LIN {X 0,Y 170.395,Z 400.641,A -85,B 0,C 180,E1 -23240.523,E2 -23240.523} C_VEL
LIN {X 0,Y 173.665,Z 396.703,A -85,B 0,C 180,E1 -23242.047,E2 -23242.047} C_VEL
LIN {X 0,Y 175.029,Z 394.829,A -85,B 0,C 180,E1 -23242.551,E2 -23242.551} C_VEL
LIN {X 0,Y 176.798,Z 393.099,A -85,B 0,C 180,E1 -23243.423,E2 -23243.423} C_VEL
LIN {X 0,Y 178.535,Z 391.866,A -85,B 0,C 180,E1 -23244.414,E2 -23244.414} C_VEL
LIN {X 0,Y 181.801,Z 388.149,A -85,B 0,C 180,E1 -23245.779,E2 -23245.779} C_VEL
LIN {X 0,Y 185.617,Z 382.76,A -85,B 0,C 180,E1 -23247.024,E2 -23247.024} C_VEL
LIN {X 0,Y 188.526,Z 380.586,A -85,B 0,C 180,E1 -23248.379,E2 -23248.379} C_VEL
LIN {X 0,Y 191.312,Z 377.501,A -85,B 0,C 180,E1 -23249.395,E2 -23249.395} C_VEL
LIN {X 0,Y 192.302,Z 378.568,A -85,B 0,C 180,E1 -23250.142,E2 -23250.142} C_VEL
LIN {X 0,Y 194.191,Z 381.489,A -85,B 0,C 180,E1 -23251.653,E2 -23251.653} C_VEL
LIN {X 0,Y 197.755,Z 388.389,A -85,B 0,C 180,E1 -23254.655,E2 -23254.655} C_VEL
LIN {X 0,Y 201.159,Z 397.142,A -85,B 0,C 180,E1 -23257.878,E2 -23257.878} C_VEL
LIN {X 0,Y 202.808,Z 403.388,A -85,B 0,C 180,E1 -23259.875,E2 -23259.875} C_VEL
LIN {X 0,Y 204.423,Z 413.612,A -85,B 0,C 180,E1 -23262.894,E2 -23262.894} C_VEL
LIN {X 0,Y 204.93,Z 420.786,A -85,B 0,C 180,E1 -23264.939,E2 -23264.939} C_VEL
LIN {X 0,Y 203.024,Z 426.169,A -85,B 0,C 180,E1 -23265.89,E2 -23265.89} C_VEL
LIN {X 0,Y 197.868,Z 437.857,A -85,B 0,C 180,E1 -23268.105,E2 -23268.105} C_VEL
LIN {X 0,Y 192.442,Z 449.393,A -85,B 0,C 180,E1 -23270.951,E2 -23270.951} C_VEL
LIN {X 0,Y 187.443,Z 458.742,A -85,B 0,C 180,E1 -23273.805,E2 -23273.805} C_VEL
LIN {X 0,Y 182.067,Z 467.908,A -85,B 0,C 180,E1 -23277.287,E2 -23277.287} C_VEL
LIN {X 0,Y 177.674,Z 475.04,A -85,B 0,C 180,E1 -23280.707,E2 -23280.707} C_VEL
LIN {X 0,Y 173.336,Z 481.783,A -85,B 0,C 180,E1 -23284.803,E2 -23284.803} C_VEL
LIN {X 0,Y 169.548,Z 487.52,A -85,B 0,C 180,E1 -23289.369,E2 -23289.369} C_VEL
LIN {X 0,Y 167.331,Z 490.895,A -85,B 0,C 180,E1 -23292.902,E2 -23292.902} C_VEL
LIN {X 0,Y 165.148,Z 494.321,A -85,B 0,C 180,E1 -23297.714,E2 -23297.714} C_VEL
LIN {X 0,Y 163.712,Z 496.576,A -85,B 0,C 180,E1 -23302.6,E2 -23302.6} C_VEL
LIN {X 0,Y 163.282,Z 497.693,A -85,B 0,C 180,E1 -23307.533,E2 -23307.533} C_VEL
LIN {X 0,Y 163.275,Z 497.703,A -85,B 0,C 180,E1 -23312.466,E2 -23312.466} C_VEL
LIN {X 0,Y 163.704,Z 496.623,A -85,B 0,C 180,E1 -23317.399,E2 -23317.399} C_VEL
LIN {X 0,Y 165.146,Z 494.408,A -85,B 0,C 180,E1 -23322.285,E2 -23322.285} C_VEL
LIN {X 0,Y 167.303,Z 491.033,A -85,B 0,C 180,E1 -23327.1,E2 -23327.1} C_VEL
LIN {X 0,Y 170.374,Z 486.387,A -85,B 0,C 180,E1 -23331.792,E2 -23331.792} C_VEL
LIN {X 0,Y 174.38,Z 480.335,A -85,B 0,C 180,E1 -23336.316,E2 -23336.316} C_VEL
LIN {X 0,Y 179.185,Z 472.711,A -85,B 0,C 180,E1 -23340.656,E2 -23340.656} C_VEL
LIN {X 0,Y 184.211,Z 464.543,A -85,B 0,C 180,E1 -23344.245,E2 -23344.245} C_VEL
LIN {X 0,Y 189.02,Z 456.226,A -85,B 0,C 180,E1 -23347.17,E2 -23347.17} C_VEL
LIN {X 0,Y 193.966,Z 446.388,A -85,B 0,C 180,E1 -23350.026,E2 -23350.026} C_VEL
LIN {X 0,Y 199.084,Z 435.684,A -85,B 0,C 180,E1 -23352.465,E2 -23352.465} C_VEL
LIN {X 0,Y 204.181,Z 423.507,A -85,B 0,C 180,E1 -23354.703,E2 -23354.703} C_VEL
LIN {X 0,Y 205.046,Z 421.302,A -85,B 0,C 180,E1 -23355.069,E2 -23355.069} C_VEL
LIN {X 0,Y 204.217,Z 411.475,A -85,B 0,C 180,E1 -23357.891,E2 -23357.891} C_VEL
LIN {X 0,Y 202.607,Z 401.977,A -85,B 0,C 180,E1 -23360.723,E2 -23360.723} C_VEL
LIN {X 0,Y 200.157,Z 394.203,A -85,B 0,C 180,E1 -23363.351,E2 -23363.351} C_VEL
LIN {X 0,Y 196.807,Z 386.307,A -85,B 0,C 180,E1 -23366.392,E2 -23366.392} C_VEL
LIN {X 0,Y 192.765,Z 378.593,A -85,B 0,C 180,E1 -23369.854,E2 -23369.854} C_VEL
LIN {X 0,Y 190.142,Z 374.291,A -85,B 0,C 180,E1 -23372.108,E2 -23372.108} C_VEL
LIN {X 0,Y 187.528,Z 370.233,A -85,B 0,C 180,E1 -23374.47,E2 -23374.47} C_VEL
LIN {X 0,Y 184.923,Z 366.507,A -85,B 0,C 180,E1 -23376.925,E2 -23376.925} C_VEL
LIN {X 0,Y 181.303,Z 361.808,A -85,B 0,C 180,E1 -23380.762,E2 -23380.762} C_VEL
LIN {X 0,Y 180.611,Z 360.907,A -85,B 0,C 180,E1 -23381.569,E2 -23381.569} C_VEL
LIN {X 0,Y 177.684,Z 357.905,A -85,B 0,C 180,E1 -23385.395,E2 -23385.395} C_VEL
LIN {X 0,Y 176.515,Z 356.153,A -85,B 0,C 180,E1 -23387.35,E2 -23387.35} C_VEL
LIN {X 0,Y 173.441,Z 353.702,A -85,B 0,C 180,E1 -23394.769,E2 -23394.769} C_VEL
LIN {X 0,Y 172.989,Z 352.533,A -85,B 0,C 180,E1 -23400,E2 -23400} C_VEL
LIN {X 0,Y 173.415,Z 354.005,A -85,B 0,C 180,E1 -23404.358,E2 -23404.358} C_VEL
LIN {X 0,Y 174.867,Z 356.398,A -85,B 0,C 180,E1 -23408.959,E2 -23408.959} C_VEL
LIN {X 0,Y 180.203,Z 363.117,A -85,B 0,C 180,E1 -23417.227,E2 -23417.227} C_VEL
LIN {X 0,Y 184.582,Z 369.399,A -85,B 0,C 180,E1 -23421.791,E2 -23421.791} C_VEL
LIN {X 0,Y 185.973,Z 371.104,A -85,B 0,C 180,E1 -23423.01,E2 -23423.01} C_VEL
LIN {X 0,Y 189.761,Z 377.14,A -85,B 0,C 180,E1 -23426.165,E2 -23426.165} C_VEL
LIN {X 0,Y 192.816,Z 383.748,A -85,B 0,C 180,E1 -23428.697,E2 -23428.697} C_VEL
LIN {X 0,Y 196.981,Z 393.192,A -85,B 0,C 180,E1 -23432.003,E2 -23432.003} C_VEL
LIN {X 0,Y 200.844,Z 404.054,A -85,B 0,C 180,E1 -23435.266,E2 -23435.266} C_VEL
LIN {X 0,Y 203.623,Z 413.079,A -85,B 0,C 180,E1 -23437.778,E2 -23437.778} C_VEL
LIN {X 0,Y 203.883,Z 414.052,A -85,B 0,C 180,E1 -23438.035,E2 -23438.035} C_VEL
LIN {X 0,Y 203.122,Z 424.995,A -85,B 0,C 180,E1 -23439.842,E2 -23439.842} C_VEL
LIN {X 0,Y 201.003,Z 438.001,A -85,B 0,C 180,E1 -23442.057,E2 -23442.057} C_VEL
LIN {X 0,Y 197.863,Z 451.759,A -85,B 0,C 180,E1 -23444.734,E2 -23444.734} C_VEL
LIN {X 0,Y 196.183,Z 456.998,A -85,B 0,C 180,E1 -23445.824,E2 -23445.824} C_VEL
LIN {X 0,Y 191.319,Z 467.171,A -85,B 0,C 180,E1 -23447.902,E2 -23447.902} C_VEL
LIN {X 0,Y 185.717,Z 477.999,A -85,B 0,C 180,E1 -23450.665,E2 -23450.665} C_VEL
LIN {X 0,Y 179.904,Z 488.58,A -85,B 0,C 180,E1 -23454.128,E2 -23454.128} C_VEL
LIN {X 0,Y 175.158,Z 496.844,A -85,B 0,C 180,E1 -23457.555,E2 -23457.555} C_VEL
LIN {X 0,Y 170.721,Z 504.775,A -85,B 0,C 180,E1 -23461.744,E2 -23461.744} C_VEL
LIN {X 0,Y 166.899,Z 511.637,A -85,B 0,C 180,E1 -23466.42,E2 -23466.42} C_VEL
LIN {X 0,Y 164.289,Z 517.048,A -85,B 0,C 180,E1 -23471.287,E2 -23471.287} C_VEL
LIN {X 0,Y 163.043,Z 520.188,A -85,B 0,C 180,E1 -23475.012,E2 -23475.012} C_VEL
LIN {X 0,Y 162.364,Z 523.309,A -85,B 0,C 180,E1 -23480.03,E2 -23480.03} C_VEL
LIN {X 0,Y 162.628,Z 525.227,A -85,B 0,C 180,E1 -23485.042,E2 -23485.042} C_VEL
LIN {X 0,Y 163.117,Z 525.911,A -85,B 0,C 180,E1 -23490.001,E2 -23490.001} C_VEL
LIN {X 0,Y 163.018,Z 525.868,A -85,B 0,C 180,E1 -23490.545,E2 -23490.545} C_VEL
LIN {X 0,Y 162.045,Z 525.642,A -85,B 0,C 180,E1 -23492.596,E2 -23492.596} C_VEL
LIN {X 0,Y 158.868,Z 524.667,A -85,B 0,C 180,E1 -23495.937,E2 -23495.937} C_VEL
LIN {X 0,Y 156.375,Z 523.542,A -85,B 0,C 180,E1 -23498.68,E2 -23498.68} C_VEL
LIN {X 0,Y 155.418,Z 522.492,A -85,B 0,C 180,E1 -23500.814,E2 -23500.814} C_VEL
LIN {X 0,Y 155.392,Z 522.07,A -85,B 0,C 180,E1 -23501.536,E2 -23501.536} C_VEL
LIN {X 0,Y 156.505,Z 518.577,A -85,B 0,C 180,E1 -23506.972,E2 -23506.972} C_VEL
LIN {X 0,Y 158.698,Z 513.952,A -85,B 0,C 180,E1 -23511.976,E2 -23511.976} C_VEL
LIN {X 0,Y 162.228,Z 507.689,A -85,B 0,C 180,E1 -23517.058,E2 -23517.058} C_VEL
LIN {X 0,Y 166.917,Z 500.018,A -85,B 0,C 180,E1 -23521.757,E2 -23521.757} C_VEL
LIN {X 0,Y 171.118,Z 493.067,A -85,B 0,C 180,E1 -23525.1,E2 -23525.1} C_VEL
LIN {X 0,Y 172.127,Z 491.669,A -85,B 0,C 180,E1 -23525.76,E2 -23525.76} C_VEL
LIN {X 0,Y 181.856,Z 487.267,A -85,B 0,C 180,E1 -23531.071,E2 -23531.071} C_VEL
LIN {X 0,Y 192.73,Z 482.107,A -85,B 0,C 180,E1 -23535.323,E2 -23535.323} C_VEL
LIN {X 0,Y 202.528,Z 477.239,A -85,B 0,C 180,E1 -23538.253,E2 -23538.253} C_VEL
LIN {X 0,Y 210.39,Z 473.107,A -85,B 0,C 180,E1 -23540.203,E2 -23540.203} C_VEL
LIN {X 0,Y 213.598,Z 471.144,A -85,B 0,C 180,E1 -23541.307,E2 -23541.307} C_VEL
LIN {X 0,Y 203.67,Z 473.371,A -85,B 0,C 180,E1 -23544.083,E2 -23544.083} C_VEL
LIN {X 0,Y 194.501,Z 474.582,A -85,B 0,C 180,E1 -23547.18,E2 -23547.18} C_VEL
LIN {X 0,Y 186.116,Z 474.785,A -85,B 0,C 180,E1 -23550.601,E2 -23550.601} C_VEL
LIN {X 0,Y 178.7,Z 473.926,A -85,B 0,C 180,E1 -23554.367,E2 -23554.367} C_VEL
LIN {X 0,Y 172.212,Z 471.988,A -85,B 0,C 180,E1 -23558.452,E2 -23558.452} C_VEL
LIN {X 0,Y 166.887,Z 468.896,A -85,B 0,C 180,E1 -23562.856,E2 -23562.856} C_VEL
LIN {X 0,Y 162.773,Z 464.607,A -85,B 0,C 180,E1 -23567.533,E2 -23567.533} C_VEL
LIN {X 0,Y 159.918,Z 459.04,A -85,B 0,C 180,E1 -23572.424,E2 -23572.424} C_VEL
LIN {X 0,Y 157.949,Z 452.039,A -85,B 0,C 180,E1 -23577.45,E2 -23577.45} C_VEL
LIN {X 0,Y 157.07,Z 443.407,A -85,B 0,C 180,E1 -23582.565,E2 -23582.565} C_VEL
LIN {X 0,Y 157.238,Z 434.358,A -85,B 0,C 180,E1 -23587.061,E2 -23587.061} C_VEL
LIN {X 0,Y 157.994,Z 425.622,A -85,B 0,C 180,E1 -23590.709,E2 -23590.709} C_VEL
LIN {X 0,Y 159.237,Z 414.25,A -85,B 0,C 180,E1 -23594.816,E2 -23594.816} C_VEL
LIN {X 0,Y 159.444,Z 414.477,A -85,B 0,C 180,E1 -23595.336,E2 -23595.336} C_VEL
LIN {X 0,Y 162.083,Z 412.559,A -85,B 0,C 180,E1 -23597.67,E2 -23597.67} C_VEL
LIN {X 0,Y 165.151,Z 409.197,A -85,B 0,C 180,E1 -23599.256,E2 -23599.256} C_VEL
LIN {X 0,Y 166.018,Z 408.45,A -85,B 0,C 180,E1 -23599.796,E2 -23599.796} C_VEL
LIN {X 0,Y 167.478,Z 407.611,A -85,B 0,C 180,E1 -23600.897,E2 -23600.897} C_VEL
LIN {X 0,Y 169.226,Z 406.208,A -85,B 0,C 180,E1 -23601.949,E2 -23601.949} C_VEL
LIN {X 0,Y 173.169,Z 401.939,A -85,B 0,C 180,E1 -23603.628,E2 -23603.628} C_VEL
LIN {X 0,Y 175.043,Z 399.736,A -85,B 0,C 180,E1 -23604.302,E2 -23604.302} C_VEL
LIN {X 0,Y 177.898,Z 397.57,A -85,B 0,C 180,E1 -23605.758,E2 -23605.758} C_VEL
LIN {X 0,Y 181.847,Z 393.49,A -85,B 0,C 180,E1 -23607.263,E2 -23607.263} C_VEL
LIN {X 0,Y 185.307,Z 389.01,A -85,B 0,C 180,E1 -23608.3,E2 -23608.3} C_VEL
LIN {X 0,Y 189.662,Z 385.356,A -85,B 0,C 180,E1 -23610.017,E2 -23610.017} C_VEL
LIN {X 0,Y 192.865,Z 391.675,A -85,B 0,C 180,E1 -23613.057,E2 -23613.057} C_VEL
LIN {X 0,Y 195.856,Z 399.435,A -85,B 0,C 180,E1 -23616.204,E2 -23616.204} C_VEL
LIN {X 0,Y 197.653,Z 405.99,A -85,B 0,C 180,E1 -23618.531,E2 -23618.531} C_VEL
LIN {X 0,Y 198.977,Z 415.488,A -85,B 0,C 180,E1 -23621.49,E2 -23621.49} C_VEL
LIN {X 0,Y 199.376,Z 423.016,A -85,B 0,C 180,E1 -23623.781,E2 -23623.781} C_VEL
LIN {X 0,Y 196.016,Z 431.306,A -85,B 0,C 180,E1 -23625.28,E2 -23625.28} C_VEL
LIN {X 0,Y 191.499,Z 440.994,A -85,B 0,C 180,E1 -23627.276,E2 -23627.276} C_VEL
LIN {X 0,Y 186.132,Z 451.696,A -85,B 0,C 180,E1 -23630.067,E2 -23630.067} C_VEL
LIN {X 0,Y 180.906,Z 460.799,A -85,B 0,C 180,E1 -23632.975,E2 -23632.975} C_VEL
LIN {X 0,Y 175.402,Z 469.712,A -85,B 0,C 180,E1 -23636.568,E2 -23636.568} C_VEL
LIN {X 0,Y 170.579,Z 477.088,A -85,B 0,C 180,E1 -23640.369,E2 -23640.369} C_VEL
LIN {X 0,Y 165.797,Z 483.956,A -85,B 0,C 180,E1 -23644.919,E2 -23644.919} C_VEL
LIN {X 0,Y 162.105,Z 489.322,A -85,B 0,C 180,E1 -23649.705,E2 -23649.705} C_VEL
LIN {X 0,Y 159.276,Z 493.371,A -85,B 0,C 180,E1 -23654.647,E2 -23654.647} C_VEL
LIN {X 0,Y 157.404,Z 496.196,A -85,B 0,C 180,E1 -23659.711,E2 -23659.711} C_VEL
LIN {X 0,Y 156.371,Z 497.879,A -85,B 0,C 180,E1 -23664.842,E2 -23664.842} C_VEL
LIN {X 0,Y 156.099,Z 498.454,A -85,B 0,C 180,E1 -23669.999,E2 -23669.999} C_VEL
LIN {X 0,Y 156.34,Z 497.909,A -85,B 0,C 180,E1 -23675.158,E2 -23675.158} C_VEL
LIN {X 0,Y 157.731,Z 495.79,A -85,B 0,C 180,E1 -23681.404,E2 -23681.404} C_VEL
LIN {X 0,Y 159.268,Z 493.481,A -85,B 0,C 180,E1 -23685.352,E2 -23685.352} C_VEL
LIN {X 0,Y 162.041,Z 489.486,A -85,B 0,C 180,E1 -23690.302,E2 -23690.302} C_VEL
LIN {X 0,Y 165.748,Z 484.16,A -85,B 0,C 180,E1 -23695.088,E2 -23695.088} C_VEL
LIN {X 0,Y 170.529,Z 477.335,A -85,B 0,C 180,E1 -23699.64,E2 -23699.64} C_VEL
LIN {X 0,Y 175.325,Z 470.019,A -85,B 0,C 180,E1 -23703.447,E2 -23703.447} C_VEL
LIN {X 0,Y 180.828,Z 461.171,A -85,B 0,C 180,E1 -23707.043,E2 -23707.043} C_VEL
LIN {X 0,Y 185.986,Z 452.109,A -85,B 0,C 180,E1 -23709.97,E2 -23709.97} C_VEL
LIN {X 0,Y 191.578,Z 441.094,A -85,B 0,C 180,E1 -23712.849,E2 -23712.849} C_VEL
LIN {X 0,Y 197.452,Z 428.462,A -85,B 0,C 180,E1 -23715.387,E2 -23715.387} C_VEL
LIN {X 0,Y 199.462,Z 423.47,A -85,B 0,C 180,E1 -23716.243,E2 -23716.243} C_VEL
LIN {X 0,Y 198.824,Z 413.416,A -85,B 0,C 180,E1 -23719.305,E2 -23719.305} C_VEL
LIN {X 0,Y 197.473,Z 404.835,A -85,B 0,C 180,E1 -23722.036,E2 -23722.036} C_VEL
LIN {X 0,Y 194.694,Z 395.967,A -85,B 0,C 180,E1 -23725.352,E2 -23725.352} C_VEL
LIN {X 0,Y 191.579,Z 388.713,A -85,B 0,C 180,E1 -23728.482,E2 -23728.482} C_VEL
LIN {X 0,Y 188.92,Z 383.501,A -85,B 0,C 180,E1 -23731.078,E2 -23731.078} C_VEL
LIN {X 0,Y 187.171,Z 380.381,A -85,B 0,C 180,E1 -23732.766,E2 -23732.766} C_VEL
LIN {X 0,Y 184.729,Z 376.311,A -85,B 0,C 180,E1 -23735.26,E2 -23735.26} C_VEL
LIN {X 0,Y 182.029,Z 372.145,A -85,B 0,C 180,E1 -23738.185,E2 -23738.185} C_VEL
LIN {X 0,Y 179.238,Z 368.091,A -85,B 0,C 180,E1 -23741.57,E2 -23741.57} C_VEL
LIN {X 0,Y 175.767,Z 363.946,A -85,B 0,C 180,E1 -23746.708,E2 -23746.708} C_VEL
LIN {X 0,Y 175.251,Z 363.062,A -85,B 0,C 180,E1 -23747.699,E2 -23747.699} C_VEL
LIN {X 0,Y 172.54,Z 360.765,A -85,B 0,C 180,E1 -23754.741,E2 -23754.741} C_VEL
LIN {X 0,Y 172.12,Z 359.576,A -85,B 0,C 180,E1 -23760,E2 -23760} C_VEL
LIN {X 0,Y 172.667,Z 361.362,A -85,B 0,C 180,E1 -23764.962,E2 -23764.962} C_VEL
LIN {X 0,Y 174.155,Z 363.955,A -85,B 0,C 180,E1 -23769.436,E2 -23769.436} C_VEL
LIN {X 0,Y 178.569,Z 369.783,A -85,B 0,C 180,E1 -23776.579,E2 -23776.579} C_VEL
LIN {X 0,Y 183.011,Z 376.374,A -85,B 0,C 180,E1 -23781.544,E2 -23781.544} C_VEL
LIN {X 0,Y 184.404,Z 378.627,A -85,B 0,C 180,E1 -23782.92,E2 -23782.92} C_VEL
LIN {X 0,Y 186.943,Z 382.917,A -85,B 0,C 180,E1 -23785.233,E2 -23785.233} C_VEL
LIN {X 0,Y 189.479,Z 389.053,A -85,B 0,C 180,E1 -23787.697,E2 -23787.697} C_VEL
LIN {X 0,Y 193.227,Z 398.499,A -85,B 0,C 180,E1 -23791.142,E2 -23791.142} C_VEL
LIN {X 0,Y 196.999,Z 410.323,A -85,B 0,C 180,E1 -23794.863,E2 -23794.863} C_VEL
LIN {X 0,Y 198.889,Z 417.407,A -85,B 0,C 180,E1 -23796.921,E2 -23796.921} C_VEL
LIN {X 0,Y 197.59,Z 428.862,A -85,B 0,C 180,E1 -23798.904,E2 -23798.904} C_VEL
LIN {X 0,Y 195.048,Z 441.617,A -85,B 0,C 180,E1 -23801.222,E2 -23801.222} C_VEL
LIN {X 0,Y 191.494,Z 455.167,A -85,B 0,C 180,E1 -23804.057,E2 -23804.057} C_VEL
LIN {X 0,Y 188.172,Z 462.544,A -85,B 0,C 180,E1 -23805.55,E2 -23805.55} C_VEL
LIN {X 0,Y 182.181,Z 474.009,A -85,B 0,C 180,E1 -23808.283,E2 -23808.283} C_VEL
LIN {X 0,Y 176.635,Z 483.673,A -85,B 0,C 180,E1 -23811.196,E2 -23811.196} C_VEL
LIN {X 0,Y 171.027,Z 493.203,A -85,B 0,C 180,E1 -23814.88,E2 -23814.88} C_VEL
LIN {X 0,Y 166.181,Z 501.152,A -85,B 0,C 180,E1 -23818.798,E2 -23818.798} C_VEL
LIN {X 0,Y 162.216,Z 507.78,A -85,B 0,C 180,E1 -23822.941,E2 -23822.941} C_VEL
LIN {X 0,Y 158.659,Z 514.025,A -85,B 0,C 180,E1 -23828.019,E2 -23828.019} C_VEL
LIN {X 0,Y 156.483,Z 518.627,A -85,B 0,C 180,E1 -23833.027,E2 -23833.027} C_VEL
LIN {X 0,Y 155.563,Z 521.284,A -85,B 0,C 180,E1 -23836.945,E2 -23836.945} C_VEL
LIN {X 0,Y 155.319,Z 523.803,A -85,B 0,C 180,E1 -23842.199,E2 -23842.199} C_VEL
LIN {X 0,Y 155.543,Z 524.615,A -85,B 0,C 180,E1 -23844.816,E2 -23844.816} C_VEL
LIN {X 0,Y 156.024,Z 525.301,A -85,B 0,C 180,E1 -23850.001,E2 -23850.001} C_VEL
LIN {X 0,Y 155.541,Z 524.604,A -85,B 0,C 180,E1 -23855.185,E2 -23855.185} C_VEL
LIN {X 0,Y 155.326,Z 522.668,A -85,B 0,C 180,E1 -23860.428,E2 -23860.428} C_VEL
LIN {X 0,Y 155.392,Z 522.07,A -85,B 0,C 180,E1 -23861.536,E2 -23861.536} C_VEL
LIN {X 0,Y 154.996,Z 520.875,A -85,B 0,C 180,E1 -23863.663,E2 -23863.663} C_VEL
LIN {X 0,Y 152.959,Z 518.412,A -85,B 0,C 180,E1 -23867.162,E2 -23867.162} C_VEL
LIN {X 0,Y 151.593,Z 516.124,A -85,B 0,C 180,E1 -23869.988,E2 -23869.988} C_VEL
LIN {X 0,Y 151.605,Z 514.199,A -85,B 0,C 180,E1 -23872.108,E2 -23872.108} C_VEL
LIN {X 0,Y 151.922,Z 513.521,A -85,B 0,C 180,E1 -23872.801,E2 -23872.801} C_VEL
LIN {X 0,Y 155.843,Z 507.069,A -85,B 0,C 180,E1 -23878.263,E2 -23878.263} C_VEL
LIN {X 0,Y 160.848,Z 499.4,A -85,B 0,C 180,E1 -23883.105,E2 -23883.105} C_VEL
LIN {X 0,Y 165.31,Z 492.452,A -85,B 0,C 180,E1 -23886.527,E2 -23886.527} C_VEL
LIN {X 0,Y 166.614,Z 490.676,A -85,B 0,C 180,E1 -23887.327,E2 -23887.327} C_VEL
LIN {X 0,Y 176.54,Z 486.795,A -85,B 0,C 180,E1 -23892.592,E2 -23892.592} C_VEL
LIN {X 0,Y 190.219,Z 481.051,A -85,B 0,C 180,E1 -23897.642,E2 -23897.642} C_VEL
LIN {X 0,Y 200.518,Z 476.424,A -85,B 0,C 180,E1 -23900.452,E2 -23900.452} C_VEL
LIN {X 0,Y 203.255,Z 474.912,A -85,B 0,C 180,E1 -23901.509,E2 -23901.509} C_VEL
LIN {X 0,Y 193.368,Z 476.206,A -85,B 0,C 180,E1 -23904.442,E2 -23904.442} C_VEL
LIN {X 0,Y 184.324,Z 476.492,A -85,B 0,C 180,E1 -23907.738,E2 -23907.738} C_VEL
LIN {X 0,Y 175.953,Z 475.747,A -85,B 0,C 180,E1 -23911.492,E2 -23911.492} C_VEL
LIN {X 0,Y 168.902,Z 474.014,A -85,B 0,C 180,E1 -23915.412,E2 -23915.412} C_VEL
LIN {X 0,Y 162.796,Z 471.138,A -85,B 0,C 180,E1 -23919.796,E2 -23919.796} C_VEL
LIN {X 0,Y 157.821,Z 467.105,A -85,B 0,C 180,E1 -23924.503,E2 -23924.503} C_VEL
LIN {X 0,Y 154.234,Z 461.843,A -85,B 0,C 180,E1 -23929.498,E2 -23929.498} C_VEL
LIN {X 0,Y 151.666,Z 455.248,A -85,B 0,C 180,E1 -23934.683,E2 -23934.683} C_VEL
LIN {X 0,Y 150.321,Z 447.13,A -85,B 0,C 180,E1 -23940,E2 -23940} C_VEL
LIN {X 0,Y 150.006,Z 438.52,A -85,B 0,C 180,E1 -23944.703,E2 -23944.703} C_VEL
LIN {X 0,Y 150.779,Z 427.092,A -85,B 0,C 180,E1 -23949.927,E2 -23949.927} C_VEL
LIN {X 0,Y 150.894,Z 425.499,A -85,B 0,C 180,E1 -23950.653,E2 -23950.653} C_VEL
LIN {X 0,Y 152.625,Z 424.517,A -85,B 0,C 180,E1 -23953.311,E2 -23953.311} C_VEL
LIN {X 0,Y 154.179,Z 422.989,A -85,B 0,C 180,E1 -23954.52,E2 -23954.52} C_VEL
LIN {X 0,Y 156.01,Z 420.996,A -85,B 0,C 180,E1 -23955.682,E2 -23955.682} C_VEL
LIN {X 0,Y 160.001,Z 418.225,A -85,B 0,C 180,E1 -23958.989,E2 -23958.989} C_VEL
LIN {X 0,Y 164.425,Z 414.134,A -85,B 0,C 180,E1 -23961.304,E2 -23961.304} C_VEL
LIN {X 0,Y 167.975,Z 411.675,A -85,B 0,C 180,E1 -23963.422,E2 -23963.422} C_VEL
LIN {X 0,Y 171.481,Z 408.304,A -85,B 0,C 180,E1 -23964.84,E2 -23964.84} C_VEL
LIN {X 0,Y 174.064,Z 405.509,A -85,B 0,C 180,E1 -23965.725,E2 -23965.725} C_VEL
LIN {X 0,Y 177.176,Z 403.17,A -85,B 0,C 180,E1 -23967.14,E2 -23967.14} C_VEL
LIN {X 0,Y 180.255,Z 400.368,A -85,B 0,C 180,E1 -23968.267,E2 -23968.267} C_VEL
LIN {X 0,Y 186.12,Z 393.925,A -85,B 0,C 180,E1 -23970.022,E2 -23970.022} C_VEL
LIN {X 0,Y 187.208,Z 393.188,A -85,B 0,C 180,E1 -23970.452,E2 -23970.452} C_VEL
LIN {X 0,Y 190.045,Z 400.104,A -85,B 0,C 180,E1 -23973.691,E2 -23973.691} C_VEL
LIN {X 0,Y 192.064,Z 406.762,A -85,B 0,C 180,E1 -23976.387,E2 -23976.387} C_VEL
LIN {X 0,Y 193.033,Z 411.991,A -85,B 0,C 180,E1 -23978.239,E2 -23978.239} C_VEL
LIN {X 0,Y 193.8,Z 420.678,A -85,B 0,C 180,E1 -23981.096,E2 -23981.096} C_VEL
LIN {X 0,Y 193.869,Z 425.436,A -85,B 0,C 180,E1 -23982.617,E2 -23982.617} C_VEL
LIN {X 0,Y 188.922,Z 436.35,A -85,B 0,C 180,E1 -23984.645,E2 -23984.645} C_VEL
LIN {X 0,Y 183.51,Z 447.138,A -85,B 0,C 180,E1 -23987.173,E2 -23987.173} C_VEL
LIN {X 0,Y 178.054,Z 457.046,A -85,B 0,C 180,E1 -23990.103,E2 -23990.103} C_VEL
LIN {X 0,Y 171.971,Z 466.719,A -85,B 0,C 180,E1 -23993.659,E2 -23993.659} C_VEL
LIN {X 0,Y 165.884,Z 475.616,A -85,B 0,C 180,E1 -23997.924,E2 -23997.924} C_VEL
LIN {X 0,Y 160.639,Z 483,A -85,B 0,C 180,E1 -24002.652,E2 -24002.652} C_VEL
LIN {X 0,Y 156.379,Z 488.737,A -85,B 0,C 180,E1 -24007.541,E2 -24007.541} C_VEL
LIN {X 0,Y 153.852,Z 492.114,A -85,B 0,C 180,E1 -24011.351,E2 -24011.351} C_VEL
LIN {X 0,Y 151.34,Z 495.539,A -85,B 0,C 180,E1 -24016.573,E2 -24016.573} C_VEL
LIN {X 0,Y 149.707,Z 497.792,A -85,B 0,C 180,E1 -24021.903,E2 -24021.903} C_VEL
LIN {X 0,Y 149.14,Z 498.911,A -85,B 0,C 180,E1 -24027.298,E2 -24027.298} C_VEL
LIN {X 0,Y 149.131,Z 498.921,A -85,B 0,C 180,E1 -24032.701,E2 -24032.701} C_VEL
LIN {X 0,Y 149.7,Z 497.837,A -85,B 0,C 180,E1 -24038.096,E2 -24038.096} C_VEL
LIN {X 0,Y 151.338,Z 495.624,A -85,B 0,C 180,E1 -24043.426,E2 -24043.426} C_VEL
LIN {X 0,Y 153.823,Z 492.248,A -85,B 0,C 180,E1 -24048.652,E2 -24048.652} C_VEL
LIN {X 0,Y 157.312,Z 487.601,A -85,B 0,C 180,E1 -24053.708,E2 -24053.708} C_VEL
LIN {X 0,Y 161.814,Z 481.546,A -85,B 0,C 180,E1 -24058.539,E2 -24058.539} C_VEL
LIN {X 0,Y 167.148,Z 473.921,A -85,B 0,C 180,E1 -24063.134,E2 -24063.134} C_VEL
LIN {X 0,Y 172.687,Z 465.749,A -85,B 0,C 180,E1 -24066.89,E2 -24066.89} C_VEL
LIN {X 0,Y 178.827,Z 455.874,A -85,B 0,C 180,E1 -24070.425,E2 -24070.425} C_VEL
LIN {X 0,Y 184.341,Z 445.784,A -85,B 0,C 180,E1 -24073.333,E2 -24073.333} C_VEL
LIN {X 0,Y 189.926,Z 434.773,A -85,B 0,C 180,E1 -24075.803,E2 -24075.803} C_VEL
LIN {X 0,Y 193.856,Z 425.949,A -85,B 0,C 180,E1 -24077.423,E2 -24077.423} C_VEL
LIN {X 0,Y 193.796,Z 419.046,A -85,B 0,C 180,E1 -24079.602,E2 -24079.602} C_VEL
LIN {X 0,Y 192.956,Z 410.612,A -85,B 0,C 180,E1 -24082.405,E2 -24082.405} C_VEL
LIN {X 0,Y 191.112,Z 403.145,A -85,B 0,C 180,E1 -24085.25,E2 -24085.25} C_VEL
LIN {X 0,Y 188.899,Z 396.826,A -85,B 0,C 180,E1 -24087.983,E2 -24087.983} C_VEL
LIN {X 0,Y 186.558,Z 391.284,A -85,B 0,C 180,E1 -24090.677,E2 -24090.677} C_VEL
LIN {X 0,Y 184.627,Z 387.32,A -85,B 0,C 180,E1 -24092.82,E2 -24092.82} C_VEL
LIN {X 0,Y 181.779,Z 382.31,A -85,B 0,C 180,E1 -24096.049,E2 -24096.049} C_VEL
LIN {X 0,Y 179.556,Z 378.481,A -85,B 0,C 180,E1 -24098.855,E2 -24098.855} C_VEL
LIN {X 0,Y 176.7,Z 374.141,A -85,B 0,C 180,E1 -24102.792,E2 -24102.792} C_VEL
LIN {X 0,Y 174.037,Z 370.51,A -85,B 0,C 180,E1 -24107.39,E2 -24107.39} C_VEL
LIN {X 0,Y 173.463,Z 369.759,A -85,B 0,C 180,E1 -24108.608,E2 -24108.608} C_VEL
LIN {X 0,Y 171.336,Z 367.673,A -85,B 0,C 180,E1 -24115.294,E2 -24115.294} C_VEL
LIN {X 0,Y 171.083,Z 366.622,A -85,B 0,C 180,E1 -24120,E2 -24120} C_VEL
LIN {X 0,Y 171.835,Z 368.822,A -85,B 0,C 180,E1 -24125.868,E2 -24125.868} C_VEL
LIN {X 0,Y 173.59,Z 372.102,A -85,B 0,C 180,E1 -24130.718,E2 -24130.718} C_VEL
LIN {X 0,Y 176.699,Z 376.283,A -85,B 0,C 180,E1 -24135.869,E2 -24135.869} C_VEL
LIN {X 0,Y 181.477,Z 383.999,A -85,B 0,C 180,E1 -24141.7,E2 -24141.7} C_VEL
LIN {X 0,Y 183.969,Z 388.732,A -85,B 0,C 180,E1 -24144.341,E2 -24144.341} C_VEL
LIN {X 0,Y 186.316,Z 395.106,A -85,B 0,C 180,E1 -24146.989,E2 -24146.989} C_VEL
LIN {X 0,Y 189.217,Z 403.168,A -85,B 0,C 180,E1 -24150.094,E2 -24150.094} C_VEL
LIN {X 0,Y 192.629,Z 415.284,A -85,B 0,C 180,E1 -24154.09,E2 -24154.09} C_VEL
LIN {X 0,Y 193.868,Z 420.718,A -85,B 0,C 180,E1 -24155.771,E2 -24155.771} C_VEL
LIN {X 0,Y 192.158,Z 432.203,A -85,B 0,C 180,E1 -24157.858,E2 -24157.858} C_VEL
LIN {X 0,Y 189.077,Z 445.232,A -85,B 0,C 180,E1 -24160.361,E2 -24160.361} C_VEL
LIN {X 0,Y 185.583,Z 457.026,A -85,B 0,C 180,E1 -24162.973,E2 -24162.973} C_VEL
LIN {X 0,Y 179.913,Z 467.923,A -85,B 0,C 180,E1 -24165.321,E2 -24165.321} C_VEL
LIN {X 0,Y 173.903,Z 478.425,A -85,B 0,C 180,E1 -24168.179,E2 -24168.179} C_VEL
LIN {X 0,Y 168.452,Z 487.354,A -85,B 0,C 180,E1 -24171.258,E2 -24171.258} C_VEL
LIN {X 0,Y 162.987,Z 495.949,A -85,B 0,C 180,E1 -24175.012,E2 -24175.012} C_VEL
LIN {X 0,Y 158.159,Z 503.541,A -85,B 0,C 180,E1 -24179.269,E2 -24179.269} C_VEL
LIN {X 0,Y 153.812,Z 510.403,A -85,B 0,C 180,E1 -24184.274,E2 -24184.274} C_VEL
LIN {X 0,Y 150.694,Z 515.839,A -85,B 0,C 180,E1 -24189.562,E2 -24189.562} C_VEL
LIN {X 0,Y 149.182,Z 518.952,A -85,B 0,C 180,E1 -24193.581,E2 -24193.581} C_VEL
LIN {X 0,Y 148.255,Z 522.076,A -85,B 0,C 180,E1 -24199.07,E2 -24199.07} C_VEL
LIN {X 0,Y 148.445,Z 524.002,A -85,B 0,C 180,E1 -24204.567,E2 -24204.567} C_VEL
LIN {X 0,Y 148.932,Z 524.691,A -85,B 0,C 180,E1 -24210.001,E2 -24210.001} C_VEL
LIN {X 0,Y 148.435,Z 523.99,A -85,B 0,C 180,E1 -24215.434,E2 -24215.434} C_VEL
LIN {X 0,Y 148.265,Z 522.05,A -85,B 0,C 180,E1 -24220.93,E2 -24220.93} C_VEL
LIN {X 0,Y 149.2,Z 518.903,A -85,B 0,C 180,E1 -24226.418,E2 -24226.418} C_VEL
LIN {X 0,Y 151.353,Z 514.492,A -85,B 0,C 180,E1 -24231.807,E2 -24231.807} C_VEL
LIN {X 0,Y 151.922,Z 513.521,A -85,B 0,C 180,E1 -24232.801,E2 -24232.801} C_VEL
LIN {X 0,Y 152.551,Z 511.427,A -85,B 0,C 180,E1 -24234.868,E2 -24234.868} C_VEL
LIN {X 0,Y 152.152,Z 507.639,A -85,B 0,C 180,E1 -24238.318,E2 -24238.318} C_VEL
LIN {X 0,Y 152.259,Z 503.362,A -85,B 0,C 180,E1 -24241.689,E2 -24241.689} C_VEL
LIN {X 0,Y 153.637,Z 500.498,A -85,B 0,C 180,E1 -24243.554,E2 -24243.554} C_VEL
LIN {X 0,Y 158.765,Z 493.068,A -85,B 0,C 180,E1 -24247.505,E2 -24247.505} C_VEL
LIN {X 0,Y 161.461,Z 489.526,A -85,B 0,C 180,E1 -24249.136,E2 -24249.136} C_VEL
LIN {X 0,Y 171.364,Z 486.201,A -85,B 0,C 180,E1 -24254.204,E2 -24254.204} C_VEL
LIN {X 0,Y 185.511,Z 480.991,A -85,B 0,C 180,E1 -24259.262,E2 -24259.262} C_VEL
LIN {X 0,Y 190.681,Z 478.978,A -85,B 0,C 180,E1 -24260.716,E2 -24260.716} C_VEL
LIN {X 0,Y 192.825,Z 477.841,A -85,B 0,C 180,E1 -24261.713,E2 -24261.713} C_VEL
LIN {X 0,Y 183.081,Z 478.227,A -85,B 0,C 180,E1 -24264.844,E2 -24264.844} C_VEL
LIN {X 0,Y 174.118,Z 477.648,A -85,B 0,C 180,E1 -24268.351,E2 -24268.351} C_VEL
LIN {X 0,Y 166.155,Z 476.035,A -85,B 0,C 180,E1 -24272.272,E2 -24272.272} C_VEL
LIN {X 0,Y 159.165,Z 473.358,A -85,B 0,C 180,E1 -24276.585,E2 -24276.585} C_VEL
LIN {X 0,Y 153.396,Z 469.556,A -85,B 0,C 180,E1 -24281.294,E2 -24281.294} C_VEL
LIN {X 0,Y 148.975,Z 464.556,A -85,B 0,C 180,E1 -24286.357,E2 -24286.357} C_VEL
LIN {X 0,Y 145.841,Z 458.283,A -85,B 0,C 180,E1 -24291.688,E2 -24291.688} C_VEL
LIN {X 0,Y 143.776,Z 450.578,A -85,B 0,C 180,E1 -24297.198,E2 -24297.198} C_VEL
LIN {X 0,Y 142.947,Z 441.191,A -85,B 0,C 180,E1 -24302.818,E2 -24302.818} C_VEL
LIN {X 0,Y 143.001,Z 435.895,A -85,B 0,C 180,E1 -24305.641,E2 -24305.641} C_VEL
LIN {X 0,Y 144.023,Z 435.062,A -85,B 0,C 180,E1 -24308.418,E2 -24308.418} C_VEL
LIN {X 0,Y 146.668,Z 432.322,A -85,B 0,C 180,E1 -24311.051,E2 -24311.051} C_VEL
LIN {X 0,Y 150.188,Z 429.656,A -85,B 0,C 180,E1 -24314.914,E2 -24314.914} C_VEL
LIN {X 0,Y 153.744,Z 426.385,A -85,B 0,C 180,E1 -24317.286,E2 -24317.286} C_VEL
LIN {X 0,Y 156.6,Z 424.559,A -85,B 0,C 180,E1 -24319.53,E2 -24319.53} C_VEL
LIN {X 0,Y 158.558,Z 423.168,A -85,B 0,C 180,E1 -24320.769,E2 -24320.769} C_VEL
LIN {X 0,Y 160.777,Z 421.184,A -85,B 0,C 180,E1 -24321.812,E2 -24321.812} C_VEL
LIN {X 0,Y 162.78,Z 419.608,A -85,B 0,C 180,E1 -24322.866,E2 -24322.866} C_VEL
LIN {X 0,Y 166.645,Z 417.046,A -85,B 0,C 180,E1 -24324.944,E2 -24324.944} C_VEL
LIN {X 0,Y 171.658,Z 412.511,A -85,B 0,C 180,E1 -24326.767,E2 -24326.767} C_VEL
LIN {X 0,Y 174.229,Z 410.075,A -85,B 0,C 180,E1 -24327.64,E2 -24327.64} C_VEL
LIN {X 0,Y 176.375,Z 408.68,A -85,B 0,C 180,E1 -24328.566,E2 -24328.566} C_VEL
LIN {X 0,Y 181.505,Z 404.142,A -85,B 0,C 180,E1 -24330.223,E2 -24330.223} C_VEL
LIN {X 0,Y 184.324,Z 401.193,A -85,B 0,C 180,E1 -24330.98,E2 -24330.98} C_VEL
LIN {X 0,Y 185.998,Z 405.844,A -85,B 0,C 180,E1 -24333.224,E2 -24333.224} C_VEL
LIN {X 0,Y 187.696,Z 412.789,A -85,B 0,C 180,E1 -24336.139,E2 -24336.139} C_VEL
LIN {X 0,Y 188.367,Z 419.895,A -85,B 0,C 180,E1 -24338.679,E2 -24338.679} C_VEL
LIN {X 0,Y 188.491,Z 426.763,A -85,B 0,C 180,E1 -24341.03,E2 -24341.03} C_VEL
LIN {X 0,Y 188.408,Z 427.875,A -85,B 0,C 180,E1 -24341.377,E2 -24341.377} C_VEL
LIN {X 0,Y 182.411,Z 440.086,A -85,B 0,C 180,E1 -24343.746,E2 -24343.746} C_VEL
LIN {X 0,Y 176.454,Z 451.209,A -85,B 0,C 180,E1 -24346.602,E2 -24346.602} C_VEL
LIN {X 0,Y 170.8,Z 460.558,A -85,B 0,C 180,E1 -24349.603,E2 -24349.603} C_VEL
LIN {X 0,Y 164.593,Z 469.731,A -85,B 0,C 180,E1 -24353.287,E2 -24353.287} C_VEL
LIN {X 0,Y 159.707,Z 476.495,A -85,B 0,C 180,E1 -24356.732,E2 -24356.732} C_VEL
LIN {X 0,Y 154.37,Z 483.611,A -85,B 0,C 180,E1 -24361.442,E2 -24361.442} C_VEL
LIN {X 0,Y 149.868,Z 489.346,A -85,B 0,C 180,E1 -24366.508,E2 -24366.508} C_VEL
LIN {X 0,Y 147.168,Z 492.722,A -85,B 0,C 180,E1 -24370.47,E2 -24370.47} C_VEL
LIN {X 0,Y 144.451,Z 496.15,A -85,B 0,C 180,E1 -24375.92,E2 -24375.92} C_VEL
LIN {X 0,Y 142.715,Z 498.4,A -85,B 0,C 180,E1 -24381.504,E2 -24381.504} C_VEL
LIN {X 0,Y 142.069,Z 499.52,A -85,B 0,C 180,E1 -24387.164,E2 -24387.164} C_VEL
LIN {X 0,Y 142.059,Z 499.529,A -85,B 0,C 180,E1 -24392.835,E2 -24392.835} C_VEL
LIN {X 0,Y 142.709,Z 498.445,A -85,B 0,C 180,E1 -24398.495,E2 -24398.495} C_VEL
LIN {X 0,Y 144.45,Z 496.233,A -85,B 0,C 180,E1 -24404.079,E2 -24404.079} C_VEL
LIN {X 0,Y 147.136,Z 492.855,A -85,B 0,C 180,E1 -24409.533,E2 -24409.533} C_VEL
LIN {X 0,Y 150.853,Z 488.208,A -85,B 0,C 180,E1 -24414.79,E2 -24414.79} C_VEL
LIN {X 0,Y 154.303,Z 483.808,A -85,B 0,C 180,E1 -24418.57,E2 -24418.57} C_VEL
LIN {X 0,Y 159.934,Z 476.359,A -85,B 0,C 180,E1 -24423.504,E2 -24423.504} C_VEL
LIN {X 0,Y 166.236,Z 467.635,A -85,B 0,C 180,E1 -24427.807,E2 -24427.807} C_VEL
LIN {X 0,Y 172.576,Z 458.03,A -85,B 0,C 180,E1 -24431.434,E2 -24431.434} C_VEL
LIN {X 0,Y 178.241,Z 448.184,A -85,B 0,C 180,E1 -24434.417,E2 -24434.417} C_VEL
LIN {X 0,Y 184.539,Z 436.426,A -85,B 0,C 180,E1 -24437.148,E2 -24437.148} C_VEL
LIN {X 0,Y 188.302,Z 428.446,A -85,B 0,C 180,E1 -24438.68,E2 -24438.68} C_VEL
LIN {X 0,Y 188.602,Z 426.226,A -85,B 0,C 180,E1 -24439.322,E2 -24439.322} C_VEL
LIN {X 0,Y 188.268,Z 416.784,A -85,B 0,C 180,E1 -24442.599,E2 -24442.599} C_VEL
LIN {X 0,Y 187.546,Z 411.733,A -85,B 0,C 180,E1 -24444.49,E2 -24444.49} C_VEL
LIN {X 0,Y 185.42,Z 403.71,A -85,B 0,C 180,E1 -24447.951,E2 -24447.951} C_VEL
LIN {X 0,Y 182.939,Z 397.071,A -85,B 0,C 180,E1 -24451.3,E2 -24451.3} C_VEL
LIN {X 0,Y 181.341,Z 393.357,A -85,B 0,C 180,E1 -24453.408,E2 -24453.408} C_VEL
LIN {X 0,Y 178.703,Z 388.261,A -85,B 0,C 180,E1 -24456.841,E2 -24456.841} C_VEL
LIN {X 0,Y 176.772,Z 384.612,A -85,B 0,C 180,E1 -24459.642,E2 -24459.642} C_VEL
LIN {X 0,Y 174.556,Z 380.766,A -85,B 0,C 180,E1 -24463.228,E2 -24463.228} C_VEL
LIN {X 0,Y 172.161,Z 377.166,A -85,B 0,C 180,E1 -24467.923,E2 -24467.923} C_VEL
LIN {X 0,Y 170.75,Z 375.545,A -85,B 0,C 180,E1 -24471.717,E2 -24471.717} C_VEL
LIN {X 0,Y 169.779,Z 373.624,A -85,B 0,C 180,E1 -24480,E2 -24480} C_VEL
LIN {X 0,Y 170.489,Z 375.922,A -85,B 0,C 180,E1 -24485.915,E2 -24485.915} C_VEL
LIN {X 0,Y 172.615,Z 379.995,A -85,B 0,C 180,E1 -24491.746,E2 -24491.746} C_VEL
LIN {X 0,Y 174.717,Z 382.993,A -85,B 0,C 180,E1 -24495.366,E2 -24495.366} C_VEL
LIN {X 0,Y 178.972,Z 390.437,A -85,B 0,C 180,E1 -24501.132,E2 -24501.132} C_VEL
LIN {X 0,Y 180.821,Z 394.363,A -85,B 0,C 180,E1 -24503.401,E2 -24503.401} C_VEL
LIN {X 0,Y 182.914,Z 400.945,A -85,B 0,C 180,E1 -24506.222,E2 -24506.222} C_VEL
LIN {X 0,Y 185.466,Z 409.215,A -85,B 0,C 180,E1 -24509.513,E2 -24509.513} C_VEL
LIN {X 0,Y 187.768,Z 418.717,A -85,B 0,C 180,E1 -24512.834,E2 -24512.834} C_VEL
LIN {X 0,Y 188.88,Z 423.966,A -85,B 0,C 180,E1 -24514.571,E2 -24514.571} C_VEL
LIN {X 0,Y 187.055,Z 433.922,A -85,B 0,C 180,E1 -24516.463,E2 -24516.463} C_VEL
LIN {X 0,Y 183.498,Z 447.242,A -85,B 0,C 180,E1 -24519.143,E2 -24519.143} C_VEL
LIN {X 0,Y 180.09,Z 457.698,A -85,B 0,C 180,E1 -24521.561,E2 -24521.561} C_VEL
LIN {X 0,Y 173.846,Z 469.207,A -85,B 0,C 180,E1 -24524.146,E2 -24524.146} C_VEL
LIN {X 0,Y 167.629,Z 479.445,A -85,B 0,C 180,E1 -24527.056,E2 -24527.056} C_VEL
LIN {X 0,Y 161.135,Z 489.468,A -85,B 0,C 180,E1 -24530.771,E2 -24530.771} C_VEL
LIN {X 0,Y 154.773,Z 498.892,A -85,B 0,C 180,E1 -24535.417,E2 -24535.417} C_VEL
LIN {X 0,Y 149.509,Z 506.545,A -85,B 0,C 180,E1 -24540.425,E2 -24540.425} C_VEL
LIN {X 0,Y 145.479,Z 512.66,A -85,B 0,C 180,E1 -24545.756,E2 -24545.756} C_VEL
LIN {X 0,Y 142.78,Z 517.392,A -85,B 0,C 180,E1 -24551.341,E2 -24551.341} C_VEL
LIN {X 0,Y 141.57,Z 520.047,A -85,B 0,C 180,E1 -24555.629,E2 -24555.629} C_VEL
LIN {X 0,Y 141.115,Z 522.57,A -85,B 0,C 180,E1 -24561.408,E2 -24561.408} C_VEL
LIN {X 0,Y 141.348,Z 523.389,A -85,B 0,C 180,E1 -24564.294,E2 -24564.294} C_VEL
LIN {X 0,Y 141.84,Z 524.081,A -85,B 0,C 180,E1 -24570.001,E2 -24570.001} C_VEL
LIN {X 0,Y 141.349,Z 523.378,A -85,B 0,C 180,E1 -24575.708,E2 -24575.708} C_VEL
LIN {X 0,Y 141.231,Z 521.433,A -85,B 0,C 180,E1 -24581.482,E2 -24581.482} C_VEL
LIN {X 0,Y 142.313,Z 518.284,A -85,B 0,C 180,E1 -24587.236,E2 -24587.236} C_VEL
LIN {X 0,Y 144.984,Z 513.4,A -85,B 0,C 180,E1 -24593.372,E2 -24593.372} C_VEL
LIN {X 0,Y 148.395,Z 508.108,A -85,B 0,C 180,E1 -24598.269,E2 -24598.269} C_VEL
LIN {X 0,Y 153.637,Z 500.498,A -85,B 0,C 180,E1 -24603.554,E2 -24603.554} C_VEL
LIN {X 0,Y 154.431,Z 498.546,A -85,B 0,C 180,E1 -24604.81,E2 -24604.81} C_VEL
LIN {X 0,Y 154.08,Z 492.001,A -85,B 0,C 180,E1 -24609.209,E2 -24609.209} C_VEL
LIN {X 0,Y 155.196,Z 489.739,A -85,B 0,C 180,E1 -24610.354,E2 -24610.354} C_VEL
LIN {X 0,Y 156.499,Z 488.289,A -85,B 0,C 180,E1 -24611.055,E2 -24611.055} C_VEL
LIN {X 0,Y 166.341,Z 485.464,A -85,B 0,C 180,E1 -24615.912,E2 -24615.912} C_VEL
LIN {X 0,Y 180.96,Z 480.805,A -85,B 0,C 180,E1 -24620.965,E2 -24620.965} C_VEL
LIN {X 0,Y 182.372,Z 479.996,A -85,B 0,C 180,E1 -24621.933,E2 -24621.933} C_VEL
LIN {X 0,Y 172.709,Z 479.516,A -85,B 0,C 180,E1 -24625.271,E2 -24625.271} C_VEL
LIN {X 0,Y 163.556,Z 477.918,A -85,B 0,C 180,E1 -24629.25,E2 -24629.25} C_VEL
LIN {X 0,Y 156.186,Z 475.477,A -85,B 0,C 180,E1 -24633.258,E2 -24633.258} C_VEL
LIN {X 0,Y 149.58,Z 471.869,A -85,B 0,C 180,E1 -24637.922,E2 -24637.922} C_VEL
LIN {X 0,Y 144.196,Z 467.126,A -85,B 0,C 180,E1 -24642.997,E2 -24642.997} C_VEL
LIN {X 0,Y 140.336,Z 461.165,A -85,B 0,C 180,E1 -24648.445,E2 -24648.445} C_VEL
LIN {X 0,Y 137.568,Z 453.852,A -85,B 0,C 180,E1 -24654.136,E2 -24654.136} C_VEL
LIN {X 0,Y 136.185,Z 445.49,A -85,B 0,C 180,E1 -24659.816,E2 -24659.816} C_VEL
LIN {X 0,Y 136.546,Z 444.61,A -85,B 0,C 180,E1 -24662.951,E2 -24662.951} C_VEL
LIN {X 0,Y 138.365,Z 442.316,A -85,B 0,C 180,E1 -24665.831,E2 -24665.831} C_VEL
LIN {X 0,Y 140.851,Z 440.049,A -85,B 0,C 180,E1 -24670.058,E2 -24670.058} C_VEL
LIN {X 0,Y 143.819,Z 437.393,A -85,B 0,C 180,E1 -24672.847,E2 -24672.847} C_VEL
LIN {X 0,Y 147.66,Z 434.669,A -85,B 0,C 180,E1 -24676.594,E2 -24676.594} C_VEL
LIN {X 0,Y 151.404,Z 431.638,A -85,B 0,C 180,E1 -24678.962,E2 -24678.962} C_VEL
LIN {X 0,Y 154.758,Z 429.599,A -85,B 0,C 180,E1 -24681.303,E2 -24681.303} C_VEL
LIN {X 0,Y 156.696,Z 428.295,A -85,B 0,C 180,E1 -24682.41,E2 -24682.41} C_VEL
LIN {X 0,Y 159.009,Z 426.362,A -85,B 0,C 180,E1 -24683.44,E2 -24683.44} C_VEL
LIN {X 0,Y 165.264,Z 422.291,A -85,B 0,C 180,E1 -24686.52,E2 -24686.52} C_VEL
LIN {X 0,Y 170.479,Z 417.926,A -85,B 0,C 180,E1 -24688.3,E2 -24688.3} C_VEL
LIN {X 0,Y 173.217,Z 415.509,A -85,B 0,C 180,E1 -24689.136,E2 -24689.136} C_VEL
LIN {X 0,Y 175.505,Z 414.087,A -85,B 0,C 180,E1 -24690.037,E2 -24690.037} C_VEL
LIN {X 0,Y 180.82,Z 409.723,A -85,B 0,C 180,E1 -24691.649,E2 -24691.649} C_VEL
LIN {X 0,Y 181.789,Z 411.534,A -85,B 0,C 180,E1 -24692.769,E2 -24692.769} C_VEL
LIN {X 0,Y 183.066,Z 418.612,A -85,B 0,C 180,E1 -24695.836,E2 -24695.836} C_VEL
LIN {X 0,Y 183.252,Z 425.912,A -85,B 0,C 180,E1 -24698.538,E2 -24698.538} C_VEL
LIN {X 0,Y 183.145,Z 429.661,A -85,B 0,C 180,E1 -24699.871,E2 -24699.871} C_VEL
LIN {X 0,Y 179.294,Z 437.551,A -85,B 0,C 180,E1 -24701.438,E2 -24701.438} C_VEL
LIN {X 0,Y 173.399,Z 448.347,A -85,B 0,C 180,E1 -24703.992,E2 -24703.992} C_VEL
LIN {X 0,Y 167.441,Z 458.258,A -85,B 0,C 180,E1 -24706.994,E2 -24706.994} C_VEL
LIN {X 0,Y 160.766,Z 467.936,A -85,B 0,C 180,E1 -24710.663,E2 -24710.663} C_VEL
LIN {X 0,Y 154.627,Z 476.126,A -85,B 0,C 180,E1 -24714.716,E2 -24714.716} C_VEL
LIN {X 0,Y 149.59,Z 482.541,A -85,B 0,C 180,E1 -24718.882,E2 -24718.882} C_VEL
LIN {X 0,Y 145.604,Z 487.271,A -85,B 0,C 180,E1 -24722.706,E2 -24722.706} C_VEL
LIN {X 0,Y 141.391,Z 492.31,A -85,B 0,C 180,E1 -24728.111,E2 -24728.111} C_VEL
LIN {X 0,Y 138.876,Z 495.201,A -85,B 0,C 180,E1 -24732.323,E2 -24732.323} C_VEL
LIN {X 0,Y 136.547,Z 498.025,A -85,B 0,C 180,E1 -24738.118,E2 -24738.118} C_VEL
LIN {X 0,Y 135.223,Z 499.707,A -85,B 0,C 180,E1 -24744.033,E2 -24744.033} C_VEL
LIN {X 0,Y 134.879,Z 500.279,A -85,B 0,C 180,E1 -24749.999,E2 -24749.999} C_VEL
LIN {X 0,Y 135.197,Z 499.735,A -85,B 0,C 180,E1 -24755.967,E2 -24755.967} C_VEL
LIN {X 0,Y 136.7,Z 497.913,A -85,B 0,C 180,E1 -24762.358,E2 -24762.358} C_VEL
LIN {X 0,Y 138.865,Z 495.307,A -85,B 0,C 180,E1 -24767.677,E2 -24767.677} C_VEL
LIN {X 0,Y 142.306,Z 491.308,A -85,B 0,C 180,E1 -24773.271,E2 -24773.271} C_VEL
LIN {X 0,Y 146.759,Z 485.982,A -85,B 0,C 180,E1 -24778.612,E2 -24778.612} C_VEL
LIN {X 0,Y 152.403,Z 479.154,A -85,B 0,C 180,E1 -24783.598,E2 -24783.598} C_VEL
LIN {X 0,Y 158.038,Z 471.83,A -85,B 0,C 180,E1 -24787.695,E2 -24787.695} C_VEL
LIN {X 0,Y 164.408,Z 462.974,A -85,B 0,C 180,E1 -24791.497,E2 -24791.497} C_VEL
LIN {X 0,Y 170.229,Z 453.914,A -85,B 0,C 180,E1 -24794.575,E2 -24794.575} C_VEL
LIN {X 0,Y 176.912,Z 442.395,A -85,B 0,C 180,E1 -24797.645,E2 -24797.645} C_VEL
LIN {X 0,Y 183.175,Z 430.241,A -85,B 0,C 180,E1 -24800.116,E2 -24800.116} C_VEL
LIN {X 0,Y 183.335,Z 422.392,A -85,B 0,C 180,E1 -24802.928,E2 -24802.928} C_VEL
LIN {X 0,Y 182.795,Z 416.241,A -85,B 0,C 180,E1 -24805.339,E2 -24805.339} C_VEL
LIN {X 0,Y 181.238,Z 409.169,A -85,B 0,C 180,E1 -24808.551,E2 -24808.551} C_VEL
LIN {X 0,Y 179.181,Z 402.793,A -85,B 0,C 180,E1 -24811.922,E2 -24811.922} C_VEL
LIN {X 0,Y 176.942,Z 397.319,A -85,B 0,C 180,E1 -24815.351,E2 -24815.351} C_VEL
LIN {X 0,Y 174.152,Z 391.173,A -85,B 0,C 180,E1 -24819.939,E2 -24819.939} C_VEL
LIN {X 0,Y 172.312,Z 387.52,A -85,B 0,C 180,E1 -24823.411,E2 -24823.411} C_VEL
LIN {X 0,Y 169.773,Z 383.336,A -85,B 0,C 180,E1 -24829.272,E2 -24829.272} C_VEL
LIN {X 0,Y 168.266,Z 381.568,A -85,B 0,C 180,E1 -24835.208,E2 -24835.208} C_VEL
LIN {X 0,Y 168.192,Z 380.569,A -85,B 0,C 180,E1 -24840,E2 -24840} C_VEL
LIN {X 0,Y 168.904,Z 383.083,A -85,B 0,C 180,E1 -24846.195,E2 -24846.195} C_VEL
LIN {X 0,Y 172.353,Z 389.256,A -85,B 0,C 180,E1 -24854.589,E2 -24854.589} C_VEL
LIN {X 0,Y 175.746,Z 395.672,A -85,B 0,C 180,E1 -24859.871,E2 -24859.871} C_VEL
LIN {X 0,Y 177.34,Z 399.236,A -85,B 0,C 180,E1 -24862.116,E2 -24862.116} C_VEL
LIN {X 0,Y 179.633,Z 407.553,A -85,B 0,C 180,E1 -24865.862,E2 -24865.862} C_VEL
LIN {X 0,Y 181.671,Z 415.71,A -85,B 0,C 180,E1 -24869.168,E2 -24869.168} C_VEL
LIN {X 0,Y 183.499,Z 425.091,A -85,B 0,C 180,E1 -24872.585,E2 -24872.585} C_VEL
LIN {X 0,Y 183.846,Z 427.161,A -85,B 0,C 180,E1 -24873.3,E2 -24873.3} C_VEL
LIN {X 0,Y 181.642,Z 437.225,A -85,B 0,C 180,E1 -24875.313,E2 -24875.313} C_VEL
LIN {X 0,Y 177.586,Z 450.463,A -85,B 0,C 180,E1 -24878.136,E2 -24878.136} C_VEL
LIN {X 0,Y 174.013,Z 459.837,A -85,B 0,C 180,E1 -24880.402,E2 -24880.402} C_VEL
LIN {X 0,Y 167.848,Z 470.396,A -85,B 0,C 180,E1 -24882.883,E2 -24882.883} C_VEL
LIN {X 0,Y 161.406,Z 480.339,A -85,B 0,C 180,E1 -24885.84,E2 -24885.84} C_VEL
LIN {X 0,Y 154.724,Z 490.108,A -85,B 0,C 180,E1 -24889.664,E2 -24889.664} C_VEL
LIN {X 0,Y 148.843,Z 498.271,A -85,B 0,C 180,E1 -24893.828,E2 -24893.828} C_VEL
LIN {X 0,Y 143.29,Z 505.928,A -85,B 0,C 180,E1 -24899.003,E2 -24899.003} C_VEL
LIN {X 0,Y 138.943,Z 512.042,A -85,B 0,C 180,E1 -24904.537,E2 -24904.537} C_VEL
LIN {X 0,Y 135.965,Z 516.772,A -85,B 0,C 180,E1 -24910.368,E2 -24910.368} C_VEL
LIN {X 0,Y 134.606,Z 519.428,A -85,B 0,C 180,E1 -24914.868,E2 -24914.868} C_VEL
LIN {X 0,Y 134.037,Z 521.954,A -85,B 0,C 180,E1 -24920.95,E2 -24920.95} C_VEL
LIN {X 0,Y 134.256,Z 522.786,A -85,B 0,C 180,E1 -24924.045,E2 -24924.045} C_VEL
LIN {X 0,Y 134.748,Z 523.471,A -85,B 0,C 180,E1 -24930.001,E2 -24930.001} C_VEL
LIN {X 0,Y 134.441,Z 523.274,A -85,B 0,C 180,E1 -24932.997,E2 -24932.997} C_VEL
LIN {X 0,Y 134.227,Z 522.762,A -85,B 0,C 180,E1 -24936.012,E2 -24936.012} C_VEL
LIN {X 0,Y 134.19,Z 520.814,A -85,B 0,C 180,E1 -24942.093,E2 -24942.093} C_VEL
LIN {X 0,Y 135.464,Z 517.665,A -85,B 0,C 180,E1 -24948.138,E2 -24948.138} C_VEL
LIN {X 0,Y 138.078,Z 513.253,A -85,B 0,C 180,E1 -24954.029,E2 -24954.029} C_VEL
LIN {X 0,Y 142.091,Z 507.488,A -85,B 0,C 180,E1 -24959.645,E2 -24959.645} C_VEL
LIN {X 0,Y 147.446,Z 500.22,A -85,B 0,C 180,E1 -24964.889,E2 -24964.889} C_VEL
LIN {X 0,Y 152.237,Z 493.68,A -85,B 0,C 180,E1 -24968.551,E2 -24968.551} C_VEL
LIN {X 0,Y 155.196,Z 489.739,A -85,B 0,C 180,E1 -24970.354,E2 -24970.354} C_VEL
LIN {X 0,Y 156.765,Z 488.227,A -85,B 0,C 180,E1 -24971.443,E2 -24971.443} C_VEL
LIN {X 0,Y 159.386,Z 486.711,A -85,B 0,C 180,E1 -24974.004,E2 -24974.004} C_VEL
LIN {X 0,Y 163.692,Z 484.496,A -85,B 0,C 180,E1 -24977.955,E2 -24977.955} C_VEL
LIN {X 0,Y 166.939,Z 483.196,A -85,B 0,C 180,E1 -24979.685,E2 -24979.685} C_VEL
LIN {X 0,Y 168.283,Z 482.792,A -85,B 0,C 180,E1 -24980.186,E2 -24980.186} C_VEL
LIN {X 0,Y 172.178,Z 481.723,A -85,B 0,C 180,E1 -24981.45,E2 -24981.45} C_VEL
LIN {X 0,Y 171.895,Z 481.34,A -85,B 0,C 180,E1 -24982.173,E2 -24982.173} C_VEL
LIN {X 0,Y 162.352,Z 479.951,A -85,B 0,C 180,E1 -24985.754,E2 -24985.754} C_VEL
LIN {X 0,Y 153.822,Z 477.552,A -85,B 0,C 180,E1 -24989.829,E2 -24989.829} C_VEL
LIN {X 0,Y 146.283,Z 474.121,A -85,B 0,C 180,E1 -24994.381,E2 -24994.381} C_VEL
LIN {X 0,Y 140.045,Z 469.597,A -85,B 0,C 180,E1 -24999.434,E2 -24999.434} C_VEL
LIN {X 0,Y 135.267,Z 463.898,A -85,B 0,C 180,E1 -25004.943,E2 -25004.943} C_VEL
LIN {X 0,Y 131.826,Z 456.91,A -85,B 0,C 180,E1 -25010.797,E2 -25010.797} C_VEL
LIN {X 0,Y 130.901,Z 454.406,A -85,B 0,C 180,E1 -25012.868,E2 -25012.868} C_VEL
LIN {X 0,Y 130.526,Z 454.354,A -85,B 0,C 180,E1 -25013.818,E2 -25013.818} C_VEL
LIN {X 0,Y 130.432,Z 453.236,A -85,B 0,C 180,E1 -25016.912,E2 -25016.912} C_VEL
LIN {X 0,Y 131.481,Z 451.189,A -85,B 0,C 180,E1 -25020,E2 -25020} C_VEL
LIN {X 0,Y 132.035,Z 450.146,A -85,B 0,C 180,E1 -25023.052,E2 -25023.052} C_VEL
LIN {X 0,Y 135.476,Z 446.566,A -85,B 0,C 180,E1 -25028.954,E2 -25028.954} C_VEL
LIN {X 0,Y 138.026,Z 444.548,A -85,B 0,C 180,E1 -25032.144,E2 -25032.144} C_VEL
LIN {X 0,Y 140.626,Z 442.484,A -85,B 0,C 180,E1 -25034.471,E2 -25034.471} C_VEL
LIN {X 0,Y 145.1,Z 439.532,A -85,B 0,C 180,E1 -25038.351,E2 -25038.351} C_VEL
LIN {X 0,Y 149.023,Z 436.733,A -85,B 0,C 180,E1 -25040.714,E2 -25040.714} C_VEL
LIN {X 0,Y 152.833,Z 434.533,A -85,B 0,C 180,E1 -25043.116,E2 -25043.116} C_VEL
LIN {X 0,Y 154.76,Z 433.269,A -85,B 0,C 180,E1 -25044.124,E2 -25044.124} C_VEL
LIN {X 0,Y 157.199,Z 431.415,A -85,B 0,C 180,E1 -25045.133,E2 -25045.133} C_VEL
LIN {X 0,Y 163.849,Z 427.406,A -85,B 0,C 180,E1 -25048.153,E2 -25048.153} C_VEL
LIN {X 0,Y 169.254,Z 423.206,A -85,B 0,C 180,E1 -25049.887,E2 -25049.887} C_VEL
LIN {X 0,Y 171.055,Z 421.675,A -85,B 0,C 180,E1 -25050.365,E2 -25050.365} C_VEL
LIN {X 0,Y 177.287,Z 417.343,A -85,B 0,C 180,E1 -25052.355,E2 -25052.355} C_VEL
LIN {X 0,Y 178.056,Z 421.614,A -85,B 0,C 180,E1 -25054.422,E2 -25054.422} C_VEL
LIN {X 0,Y 178.043,Z 429.383,A -85,B 0,C 180,E1 -25057.482,E2 -25057.482} C_VEL
LIN {X 0,Y 177.656,Z 432.561,A -85,B 0,C 180,E1 -25058.619,E2 -25058.619} C_VEL
LIN {X 0,Y 171.508,Z 443.87,A -85,B 0,C 180,E1 -25060.969,E2 -25060.969} C_VEL
LIN {X 0,Y 165.429,Z 454.118,A -85,B 0,C 180,E1 -25063.761,E2 -25063.761} C_VEL
LIN {X 0,Y 159.261,Z 463.22,A -85,B 0,C 180,E1 -25066.842,E2 -25066.842} C_VEL
LIN {X 0,Y 152.568,Z 472.143,A -85,B 0,C 180,E1 -25070.699,E2 -25070.699} C_VEL
LIN {X 0,Y 146.61,Z 479.524,A -85,B 0,C 180,E1 -25074.883,E2 -25074.883} C_VEL
LIN {X 0,Y 142.077,Z 484.83,A -85,B 0,C 180,E1 -25078.708,E2 -25078.708} C_VEL
LIN {X 0,Y 136.976,Z 490.566,A -85,B 0,C 180,E1 -25084.143,E2 -25084.143} C_VEL
LIN {X 0,Y 133.879,Z 493.943,A -85,B 0,C 180,E1 -25088.44,E2 -25088.44} C_VEL
LIN {X 0,Y 130.776,Z 497.367,A -85,B 0,C 180,E1 -25094.412,E2 -25094.412} C_VEL
LIN {X 0,Y 128.757,Z 499.616,A -85,B 0,C 180,E1 -25100.575,E2 -25100.575} C_VEL
LIN {X 0,Y 127.931,Z 500.738,A -85,B 0,C 180,E1 -25106.85,E2 -25106.85} C_VEL
LIN {X 0,Y 127.919,Z 500.747,A -85,B 0,C 180,E1 -25113.149,E2 -25113.149} C_VEL
LIN {X 0,Y 128.751,Z 499.659,A -85,B 0,C 180,E1 -25119.424,E2 -25119.424} C_VEL
LIN {X 0,Y 130.773,Z 497.449,A -85,B 0,C 180,E1 -25125.587,E2 -25125.587} C_VEL
LIN {X 0,Y 133.847,Z 494.073,A -85,B 0,C 180,E1 -25131.564,E2 -25131.564} C_VEL
LIN {X 0,Y 138.086,Z 489.425,A -85,B 0,C 180,E1 -25137.262,E2 -25137.262} C_VEL
LIN {X 0,Y 142.019,Z 485.022,A -85,B 0,C 180,E1 -25141.305,E2 -25141.305} C_VEL
LIN {X 0,Y 148.145,Z 477.771,A -85,B 0,C 180,E1 -25146.405,E2 -25146.405} C_VEL
LIN {X 0,Y 155.276,Z 468.844,A -85,B 0,C 180,E1 -25151.017,E2 -25151.017} C_VEL
LIN {X 0,Y 162.223,Z 459.234,A -85,B 0,C 180,E1 -25154.748,E2 -25154.748} C_VEL
LIN {X 0,Y 168.419,Z 449.382,A -85,B 0,C 180,E1 -25157.79,E2 -25157.79} C_VEL
LIN {X 0,Y 175.234,Z 437.616,A -85,B 0,C 180,E1 -25160.538,E2 -25160.538} C_VEL
LIN {X 0,Y 177.547,Z 433.126,A -85,B 0,C 180,E1 -25161.423,E2 -25161.423} C_VEL
LIN {X 0,Y 177.966,Z 432.004,A -85,B 0,C 180,E1 -25161.709,E2 -25161.709} C_VEL
LIN {X 0,Y 178.269,Z 424.936,A -85,B 0,C 180,E1 -25164.444,E2 -25164.444} C_VEL
LIN {X 0,Y 177.951,Z 420.209,A -85,B 0,C 180,E1 -25166.432,E2 -25166.432} C_VEL
LIN {X 0,Y 176.788,Z 413.811,A -85,B 0,C 180,E1 -25169.545,E2 -25169.545} C_VEL
LIN {X 0,Y 174.7,Z 406.524,A -85,B 0,C 180,E1 -25173.735,E2 -25173.735} C_VEL
LIN {X 0,Y 172.987,Z 401.904,A -85,B 0,C 180,E1 -25176.884,E2 -25176.884} C_VEL
LIN {X 0,Y 170.795,Z 396.757,A -85,B 0,C 180,E1 -25181.158,E2 -25181.158} C_VEL
LIN {X 0,Y 169.913,Z 394.732,A -85,B 0,C 180,E1 -25183.17,E2 -25183.17} C_VEL
LIN {X 0,Y 168.008,Z 391.1,A -85,B 0,C 180,E1 -25187.927,E2 -25187.927} C_VEL
LIN {X 0,Y 167.318,Z 389.786,A -85,B 0,C 180,E1 -25190.327,E2 -25190.327} C_VEL
LIN {X 0,Y 166.208,Z 388.139,A -85,B 0,C 180,E1 -25196.363,E2 -25196.363} C_VEL
LIN {X 0,Y 166.324,Z 387.444,A -85,B 0,C 180,E1 -25200,E2 -25200} C_VEL
LIN {X 0,Y 166.865,Z 389.759,A -85,B 0,C 180,E1 -25205.741,E2 -25205.741} C_VEL
LIN {X 0,Y 169.461,Z 394.947,A -85,B 0,C 180,E1 -25213.185,E2 -25213.185} C_VEL
LIN {X 0,Y 172.604,Z 401.59,A -85,B 0,C 180,E1 -25219.01,E2 -25219.01} C_VEL
LIN {X 0,Y 174.055,Z 405.036,A -85,B 0,C 180,E1 -25221.309,E2 -25221.309} C_VEL
LIN {X 0,Y 176.324,Z 415.151,A -85,B 0,C 180,E1 -25226.004,E2 -25226.004} C_VEL
LIN {X 0,Y 177.991,Z 424.215,A -85,B 0,C 180,E1 -25229.696,E2 -25229.696} C_VEL
LIN {X 0,Y 178.833,Z 430.151,A -85,B 0,C 180,E1 -25231.926,E2 -25231.926} C_VEL
LIN {X 0,Y 177.943,Z 434.539,A -85,B 0,C 180,E1 -25232.894,E2 -25232.894} C_VEL
LIN {X 0,Y 174.176,Z 446.634,A -85,B 0,C 180,E1 -25235.453,E2 -25235.453} C_VEL
LIN {X 0,Y 169.471,Z 459,A -85,B 0,C 180,E1 -25238.466,E2 -25238.466} C_VEL
LIN {X 0,Y 163.046,Z 469.788,A -85,B 0,C 180,E1 -25241.034,E2 -25241.034} C_VEL
LIN {X 0,Y 156.346,Z 479.73,A -85,B 0,C 180,E1 -25244.01,E2 -25244.01} C_VEL
LIN {X 0,Y 149.317,Z 489.495,A -85,B 0,C 180,E1 -25247.879,E2 -25247.879} C_VEL
LIN {X 0,Y 142.559,Z 498.322,A -85,B 0,C 180,E1 -25252.537,E2 -25252.537} C_VEL
LIN {X 0,Y 137.178,Z 505.313,A -85,B 0,C 180,E1 -25257.457,E2 -25257.457} C_VEL
LIN {X 0,Y 132.462,Z 511.423,A -85,B 0,C 180,E1 -25263.194,E2 -25263.194} C_VEL
LIN {X 0,Y 129.204,Z 516.154,A -85,B 0,C 180,E1 -25269.295,E2 -25269.295} C_VEL
LIN {X 0,Y 127.67,Z 518.81,A -85,B 0,C 180,E1 -25274.024,E2 -25274.024} C_VEL
LIN {X 0,Y 126.964,Z 521.338,A -85,B 0,C 180,E1 -25280.442,E2 -25280.442} C_VEL
LIN {X 0,Y 127.182,Z 522.237,A -85,B 0,C 180,E1 -25284.078,E2 -25284.078} C_VEL
LIN {X 0,Y 127.655,Z 522.861,A -85,B 0,C 180,E1 -25290.001,E2 -25290.001} C_VEL
LIN {X 0,Y 127.159,Z 522.239,A -85,B 0,C 180,E1 -25295.822,E2 -25295.822} C_VEL
LIN {X 0,Y 127.181,Z 520.196,A -85,B 0,C 180,E1 -25302.771,E2 -25302.771} C_VEL
LIN {X 0,Y 128.65,Z 517.046,A -85,B 0,C 180,E1 -25309.135,E2 -25309.135} C_VEL
LIN {X 0,Y 131.531,Z 512.633,A -85,B 0,C 180,E1 -25315.307,E2 -25315.307} C_VEL
LIN {X 0,Y 135.867,Z 506.867,A -85,B 0,C 180,E1 -25321.15,E2 -25321.15} C_VEL
LIN {X 0,Y 141.609,Z 499.602,A -85,B 0,C 180,E1 -25326.553,E2 -25326.553} C_VEL
LIN {X 0,Y 146.702,Z 493.062,A -85,B 0,C 180,E1 -25330.297,E2 -25330.297} C_VEL
LIN {X 0,Y 151.722,Z 486.893,A -85,B 0,C 180,E1 -25333.099,E2 -25333.099} C_VEL
LIN {X 0,Y 161.487,Z 484.591,A -85,B 0,C 180,E1 -25337.72,E2 -25337.72} C_VEL
LIN {X 0,Y 168.283,Z 482.792,A -85,B 0,C 180,E1 -25340.186,E2 -25340.186} C_VEL
LIN {X 0,Y 168.741,Z 482.475,A -85,B 0,C 180,E1 -25340.725,E2 -25340.725} C_VEL
LIN {X 0,Y 167.949,Z 482.093,A -85,B 0,C 180,E1 -25341.478,E2 -25341.478} C_VEL
LIN {X 0,Y 165.47,Z 481.726,A -85,B 0,C 180,E1 -25342.443,E2 -25342.443} C_VEL
LIN {X 0,Y 155.349,Z 480.487,A -85,B 0,C 180,E1 -25344.931,E2 -25344.931} C_VEL
LIN {X 0,Y 153.599,Z 480.041,A -85,B 0,C 180,E1 -25345.598,E2 -25345.598} C_VEL
LIN {X 0,Y 143.673,Z 476.324,A -85,B 0,C 180,E1 -25350.715,E2 -25350.715} C_VEL
LIN {X 0,Y 136.547,Z 471.991,A -85,B 0,C 180,E1 -25355.685,E2 -25355.685} C_VEL
LIN {X 0,Y 130.711,Z 466.535,A -85,B 0,C 180,E1 -25361.18,E2 -25361.18} C_VEL
LIN {X 0,Y 128.043,Z 462.784,A -85,B 0,C 180,E1 -25364.684,E2 -25364.684} C_VEL
LIN {X 0,Y 126.675,Z 462.275,A -85,B 0,C 180,E1 -25367.178,E2 -25367.178} C_VEL
LIN {X 0,Y 125.782,Z 459.589,A -85,B 0,C 180,E1 -25373.584,E2 -25373.584} C_VEL
LIN {X 0,Y 125.622,Z 458.541,A -85,B 0,C 180,E1 -25376.793,E2 -25376.793} C_VEL
LIN {X 0,Y 126.506,Z 456.723,A -85,B 0,C 180,E1 -25380.161,E2 -25380.161} C_VEL
LIN {X 0,Y 128.781,Z 453.9,A -85,B 0,C 180,E1 -25386.266,E2 -25386.266} C_VEL
LIN {X 0,Y 134.396,Z 449.519,A -85,B 0,C 180,E1 -25393.611,E2 -25393.611} C_VEL
LIN {X 0,Y 139.033,Z 446.385,A -85,B 0,C 180,E1 -25397.656,E2 -25397.656} C_VEL
LIN {X 0,Y 142.506,Z 444.269,A -85,B 0,C 180,E1 -25400.196,E2 -25400.196} C_VEL
LIN {X 0,Y 146.626,Z 441.654,A -85,B 0,C 180,E1 -25402.548,E2 -25402.548} C_VEL
LIN {X 0,Y 150.557,Z 439.486,A -85,B 0,C 180,E1 -25404.843,E2 -25404.843} C_VEL
LIN {X 0,Y 152.793,Z 438.12,A -85,B 0,C 180,E1 -25405.911,E2 -25405.911} C_VEL
LIN {X 0,Y 155.349,Z 436.358,A -85,B 0,C 180,E1 -25406.898,E2 -25406.898} C_VEL
LIN {X 0,Y 161.608,Z 432.857,A -85,B 0,C 180,E1 -25409.568,E2 -25409.568} C_VEL
LIN {X 0,Y 166.838,Z 429.216,A -85,B 0,C 180,E1 -25411.218,E2 -25411.218} C_VEL
LIN {X 0,Y 171.017,Z 426.065,A -85,B 0,C 180,E1 -25412.293,E2 -25412.293} C_VEL
LIN {X 0,Y 173.162,Z 425.33,A -85,B 0,C 180,E1 -25413.224,E2 -25413.224} C_VEL
LIN {X 0,Y 172.784,Z 433.24,A -85,B 0,C 180,E1 -25416.55,E2 -25416.55} C_VEL
LIN {X 0,Y 172.682,Z 434.313,A -85,B 0,C 180,E1 -25416.991,E2 -25416.991} C_VEL
LIN {X 0,Y 166.746,Z 444.808,A -85,B 0,C 180,E1 -25419.214,E2 -25419.214} C_VEL
LIN {X 0,Y 160.609,Z 454.724,A -85,B 0,C 180,E1 -25421.935,E2 -25421.935} C_VEL
LIN {X 0,Y 154.184,Z 463.825,A -85,B 0,C 180,E1 -25425.047,E2 -25425.047} C_VEL
LIN {X 0,Y 147.169,Z 472.75,A -85,B 0,C 180,E1 -25428.956,E2 -25428.956} C_VEL
LIN {X 0,Y 140.868,Z 480.134,A -85,B 0,C 180,E1 -25433.223,E2 -25433.223} C_VEL
LIN {X 0,Y 136.076,Z 485.439,A -85,B 0,C 180,E1 -25437.159,E2 -25437.159} C_VEL
LIN {X 0,Y 130.634,Z 491.176,A -85,B 0,C 180,E1 -25442.787,E2 -25442.787} C_VEL
LIN {X 0,Y 127.321,Z 494.552,A -85,B 0,C 180,E1 -25447.269,E2 -25447.269} C_VEL
LIN {X 0,Y 123.955,Z 497.978,A -85,B 0,C 180,E1 -25453.531,E2 -25453.531} C_VEL
LIN {X 0,Y 121.794,Z 500.223,A -85,B 0,C 180,E1 -25460.03,E2 -25460.03} C_VEL
LIN {X 0,Y 120.863,Z 501.347,A -85,B 0,C 180,E1 -25466.666,E2 -25466.666} C_VEL
LIN {X 0,Y 120.851,Z 501.356,A -85,B 0,C 180,E1 -25473.333,E2 -25473.333} C_VEL
LIN {X 0,Y 121.789,Z 500.266,A -85,B 0,C 180,E1 -25479.968,E2 -25479.968} C_VEL
LIN {X 0,Y 123.952,Z 498.058,A -85,B 0,C 180,E1 -25486.468,E2 -25486.468} C_VEL
LIN {X 0,Y 127.291,Z 494.68,A -85,B 0,C 180,E1 -25492.735,E2 -25492.735} C_VEL
LIN {X 0,Y 131.825,Z 490.033,A -85,B 0,C 180,E1 -25498.673,E2 -25498.673} C_VEL
LIN {X 0,Y 137.582,Z 483.971,A -85,B 0,C 180,E1 -25504.187,E2 -25504.187} C_VEL
LIN {X 0,Y 144.263,Z 476.339,A -85,B 0,C 180,E1 -25509.294,E2 -25509.294} C_VEL
LIN {X 0,Y 150.987,Z 468.162,A -85,B 0,C 180,E1 -25513.358,E2 -25513.358} C_VEL
LIN {X 0,Y 157.274,Z 459.835,A -85,B 0,C 180,E1 -25516.564,E2 -25516.564} C_VEL
LIN {X 0,Y 163.754,Z 449.98,A -85,B 0,C 180,E1 -25519.622,E2 -25519.622} C_VEL
LIN {X 0,Y 170.823,Z 438.212,A -85,B 0,C 180,E1 -25522.371,E2 -25522.371} C_VEL
LIN {X 0,Y 172.621,Z 434.865,A -85,B 0,C 180,E1 -25523.034,E2 -25523.034} C_VEL
LIN {X 0,Y 173.194,Z 429.007,A -85,B 0,C 180,E1 -25525.382,E2 -25525.382} C_VEL
LIN {X 0,Y 173.116,Z 424.39,A -85,B 0,C 180,E1 -25527.458,E2 -25527.458} C_VEL
LIN {X 0,Y 172.226,Z 418.204,A -85,B 0,C 180,E1 -25530.68,E2 -25530.68} C_VEL
LIN {X 0,Y 170.724,Z 411.886,A -85,B 0,C 180,E1 -25534.521,E2 -25534.521} C_VEL
LIN {X 0,Y 169.194,Z 407.104,A -85,B 0,C 180,E1 -25538.047,E2 -25538.047} C_VEL
LIN {X 0,Y 167.689,Z 402.957,A -85,B 0,C 180,E1 -25541.672,E2 -25541.672} C_VEL
LIN {X 0,Y 166.303,Z 399.758,A -85,B 0,C 180,E1 -25545.311,E2 -25545.311} C_VEL
LIN {X 0,Y 164.972,Z 396.63,A -85,B 0,C 180,E1 -25550.188,E2 -25550.188} C_VEL
LIN {X 0,Y 164.077,Z 395.15,A -85,B 0,C 180,E1 -25555.085,E2 -25555.085} C_VEL
LIN {X 0,Y 164.183,Z 394.219,A -85,B 0,C 180,E1 -25560,E2 -25560} C_VEL
LIN {X 0,Y 164.513,Z 396.13,A -85,B 0,C 180,E1 -25564.901,E2 -25564.901} C_VEL
LIN {X 0,Y 166.56,Z 401.002,A -85,B 0,C 180,E1 -25572.179,E2 -25572.179} C_VEL
LIN {X 0,Y 167.516,Z 403.417,A -85,B 0,C 180,E1 -25574.579,E2 -25574.579} C_VEL
LIN {X 0,Y 169.298,Z 407.396,A -85,B 0,C 180,E1 -25578.14,E2 -25578.14} C_VEL
LIN {X 0,Y 170.571,Z 410.78,A -85,B 0,C 180,E1 -25580.501,E2 -25580.501} C_VEL
LIN {X 0,Y 172.326,Z 420.826,A -85,B 0,C 180,E1 -25585.356,E2 -25585.356} C_VEL
LIN {X 0,Y 173.624,Z 431.134,A -85,B 0,C 180,E1 -25589.689,E2 -25589.689} C_VEL
LIN {X 0,Y 173.808,Z 434.094,A -85,B 0,C 180,E1 -25590.791,E2 -25590.791} C_VEL
LIN {X 0,Y 169.795,Z 446.341,A -85,B 0,C 180,E1 -25593.459,E2 -25593.459} C_VEL
LIN {X 0,Y 164.885,Z 458.483,A -85,B 0,C 180,E1 -25596.466,E2 -25596.466} C_VEL
LIN {X 0,Y 162.622,Z 462.728,A -85,B 0,C 180,E1 -25597.509,E2 -25597.509} C_VEL
LIN {X 0,Y 156.098,Z 472.719,A -85,B 0,C 180,E1 -25600.059,E2 -25600.059} C_VEL
LIN {X 0,Y 149.249,Z 482.12,A -85,B 0,C 180,E1 -25603.124,E2 -25603.124} C_VEL
LIN {X 0,Y 142.089,Z 491.38,A -85,B 0,C 180,E1 -25607.149,E2 -25607.149} C_VEL
LIN {X 0,Y 135.794,Z 499.102,A -85,B 0,C 180,E1 -25611.607,E2 -25611.607} C_VEL
LIN {X 0,Y 129.737,Z 506.354,A -85,B 0,C 180,E1 -25617.2,E2 -25617.2} C_VEL
LIN {X 0,Y 125.045,Z 512.098,A -85,B 0,C 180,E1 -25623.281,E2 -25623.281} C_VEL
LIN {X 0,Y 121.834,Z 516.48,A -85,B 0,C 180,E1 -25629.751,E2 -25629.751} C_VEL
LIN {X 0,Y 120.152,Z 519.606,A -85,B 0,C 180,E1 -25636.47,E2 -25636.47} C_VEL
LIN {X 0,Y 120.106,Z 521.689,A -85,B 0,C 180,E1 -25644.124,E2 -25644.124} C_VEL
LIN {X 0,Y 120.563,Z 522.251,A -85,B 0,C 180,E1 -25650.001,E2 -25650.001} C_VEL
LIN {X 0,Y 120.081,Z 521.692,A -85,B 0,C 180,E1 -25655.756,E2 -25655.756} C_VEL
LIN {X 0,Y 119.907,Z 520.701,A -85,B 0,C 180,E1 -25660.128,E2 -25660.128} C_VEL
LIN {X 0,Y 120.783,Z 518.151,A -85,B 0,C 180,E1 -25666.915,E2 -25666.915} C_VEL
LIN {X 0,Y 123.268,Z 514.382,A -85,B 0,C 180,E1 -25673.523,E2 -25673.523} C_VEL
LIN {X 0,Y 127.212,Z 509.306,A -85,B 0,C 180,E1 -25679.817,E2 -25679.817} C_VEL
LIN {X 0,Y 132.676,Z 502.818,A -85,B 0,C 180,E1 -25685.64,E2 -25685.64} C_VEL
LIN {X 0,Y 139.362,Z 494.711,A -85,B 0,C 180,E1 -25690.965,E2 -25690.965} C_VEL
LIN {X 0,Y 146.582,Z 486.152,A -85,B 0,C 180,E1 -25695.009,E2 -25695.009} C_VEL
LIN {X 0,Y 147.443,Z 485.36,A -85,B 0,C 180,E1 -25695.4,E2 -25695.4} C_VEL
LIN {X 0,Y 156.832,Z 483.538,A -85,B 0,C 180,E1 -25699.625,E2 -25699.625} C_VEL
LIN {X 0,Y 161.818,Z 482.446,A -85,B 0,C 180,E1 -25701.424,E2 -25701.424} C_VEL
LIN {X 0,Y 161.366,Z 481.877,A -85,B 0,C 180,E1 -25702.429,E2 -25702.429} C_VEL
LIN {X 0,Y 153.599,Z 480.041,A -85,B 0,C 180,E1 -25705.598,E2 -25705.598} C_VEL
LIN {X 0,Y 149.466,Z 478.997,A -85,B 0,C 180,E1 -25707.141,E2 -25707.141} C_VEL
LIN {X 0,Y 141.651,Z 476.937,A -85,B 0,C 180,E1 -25709.4,E2 -25709.4} C_VEL
LIN {X 0,Y 134.244,Z 474.269,A -85,B 0,C 180,E1 -25711.893,E2 -25711.893} C_VEL
LIN {X 0,Y 130.85,Z 472.327,A -85,B 0,C 180,E1 -25713.805,E2 -25713.805} C_VEL
LIN {X 0,Y 128.415,Z 470.601,A -85,B 0,C 180,E1 -25715.766,E2 -25715.766} C_VEL
LIN {X 0,Y 126.913,Z 470.398,A -85,B 0,C 180,E1 -25717.193,E2 -25717.193} C_VEL
LIN {X 0,Y 124.603,Z 469.557,A -85,B 0,C 180,E1 -25720.22,E2 -25720.22} C_VEL
LIN {X 0,Y 123.163,Z 468.226,A -85,B 0,C 180,E1 -25723.423,E2 -25723.423} C_VEL
LIN {X 0,Y 120.877,Z 466.124,A -85,B 0,C 180,E1 -25729.955,E2 -25729.955} C_VEL
LIN {X 0,Y 120.687,Z 464.74,A -85,B 0,C 180,E1 -25733.312,E2 -25733.312} C_VEL
LIN {X 0,Y 120.582,Z 463.632,A -85,B 0,C 180,E1 -25736.659,E2 -25736.659} C_VEL
LIN {X 0,Y 123.779,Z 459.213,A -85,B 0,C 180,E1 -25746.521,E2 -25746.521} C_VEL
LIN {X 0,Y 131.084,Z 453.999,A -85,B 0,C 180,E1 -25755.55,E2 -25755.55} C_VEL
LIN {X 0,Y 139.909,Z 448.855,A -85,B 0,C 180,E1 -25762.132,E2 -25762.132} C_VEL
LIN {X 0,Y 144.207,Z 446.373,A -85,B 0,C 180,E1 -25764.472,E2 -25764.472} C_VEL
LIN {X 0,Y 148.442,Z 444.176,A -85,B 0,C 180,E1 -25766.73,E2 -25766.73} C_VEL
LIN {X 0,Y 153.488,Z 441.162,A -85,B 0,C 180,E1 -25768.735,E2 -25768.735} C_VEL
LIN {X 0,Y 160.909,Z 437.15,A -85,B 0,C 180,E1 -25771.609,E2 -25771.609} C_VEL
LIN {X 0,Y 168.07,Z 432.447,A -85,B 0,C 180,E1 -25773.563,E2 -25773.563} C_VEL
LIN {X 0,Y 167.653,Z 435.982,A -85,B 0,C 180,E1 -25775.114,E2 -25775.114} C_VEL
LIN {X 0,Y 167.318,Z 437.168,A -85,B 0,C 180,E1 -25775.513,E2 -25775.513} C_VEL
LIN {X 0,Y 161.391,Z 446.968,A -85,B 0,C 180,E1 -25777.667,E2 -25777.667} C_VEL
LIN {X 0,Y 154.826,Z 456.914,A -85,B 0,C 180,E1 -25780.506,E2 -25780.506} C_VEL
LIN {X 0,Y 147.067,Z 467.131,A -85,B 0,C 180,E1 -25784.207,E2 -25784.207} C_VEL
LIN {X 0,Y 139.924,Z 475.599,A -85,B 0,C 180,E1 -25788.277,E2 -25788.277} C_VEL
LIN {X 0,Y 133.502,Z 482.621,A -85,B 0,C 180,E1 -25792.741,E2 -25792.741} C_VEL
LIN {X 0,Y 127.09,Z 489.099,A -85,B 0,C 180,E1 -25798.308,E2 -25798.308} C_VEL
LIN {X 0,Y 121.933,Z 494.138,A -85,B 0,C 180,E1 -25804.386,E2 -25804.386} C_VEL
LIN {X 0,Y 118.807,Z 497.03,A -85,B 0,C 180,E1 -25809.21,E2 -25809.21} C_VEL
LIN {X 0,Y 115.713,Z 499.978,A -85,B 0,C 180,E1 -25816.359,E2 -25816.359} C_VEL
LIN {X 0,Y 114.134,Z 501.533,A -85,B 0,C 180,E1 -25822.925,E2 -25822.925} C_VEL
LIN {X 0,Y 113.659,Z 502.104,A -85,B 0,C 180,E1 -25829.999,E2 -25829.999} C_VEL
LIN {X 0,Y 114.114,Z 501.56,A -85,B 0,C 180,E1 -25837.075,E2 -25837.075} C_VEL
LIN {X 0,Y 115.845,Z 499.912,A -85,B 0,C 180,E1 -25844.043,E2 -25844.043} C_VEL
LIN {X 0,Y 118.796,Z 497.131,A -85,B 0,C 180,E1 -25850.79,E2 -25850.79} C_VEL
LIN {X 0,Y 123.066,Z 493.131,A -85,B 0,C 180,E1 -25857.184,E2 -25857.184} C_VEL
LIN {X 0,Y 128.499,Z 487.802,A -85,B 0,C 180,E1 -25863.156,E2 -25863.156} C_VEL
LIN {X 0,Y 135.162,Z 480.976,A -85,B 0,C 180,E1 -25868.605,E2 -25868.605} C_VEL
LIN {X 0,Y 141.838,Z 473.64,A -85,B 0,C 180,E1 -25872.945,E2 -25872.945} C_VEL
LIN {X 0,Y 149.192,Z 464.776,A -85,B 0,C 180,E1 -25876.899,E2 -25876.899} C_VEL
LIN {X 0,Y 156.932,Z 454.086,A -85,B 0,C 180,E1 -25880.558,E2 -25880.558} C_VEL
LIN {X 0,Y 164.104,Z 442.985,A -85,B 0,C 180,E1 -25883.415,E2 -25883.415} C_VEL
LIN {X 0,Y 167.551,Z 437.134,A -85,B 0,C 180,E1 -25884.636,E2 -25884.636} C_VEL
LIN {X 0,Y 168.275,Z 431.363,A -85,B 0,C 180,E1 -25887.115,E2 -25887.115} C_VEL
LIN {X 0,Y 168.105,Z 425.951,A -85,B 0,C 180,E1 -25889.888,E2 -25889.888} C_VEL
LIN {X 0,Y 167.128,Z 419.451,A -85,B 0,C 180,E1 -25893.797,E2 -25893.797} C_VEL
LIN {X 0,Y 165.901,Z 414.206,A -85,B 0,C 180,E1 -25897.588,E2 -25897.588} C_VEL
LIN {X 0,Y 164.639,Z 409.929,A -85,B 0,C 180,E1 -25901.327,E2 -25901.327} C_VEL
LIN {X 0,Y 163.488,Z 406.543,A -85,B 0,C 180,E1 -25905.053,E2 -25905.053} C_VEL
LIN {X 0,Y 162.334,Z 403.374,A -85,B 0,C 180,E1 -25910.027,E2 -25910.027} C_VEL
LIN {X 0,Y 161.568,Z 401.813,A -85,B 0,C 180,E1 -25915.009,E2 -25915.009} C_VEL
LIN {X 0,Y 161.754,Z 400.937,A -85,B 0,C 180,E1 -25920,E2 -25920} C_VEL
LIN {X 0,Y 162.028,Z 402.924,A -85,B 0,C 180,E1 -25924.976,E2 -25924.976} C_VEL
LIN {X 0,Y 163.921,Z 407.925,A -85,B 0,C 180,E1 -25932.378,E2 -25932.378} C_VEL
LIN {X 0,Y 166.379,Z 414.621,A -85,B 0,C 180,E1 -25938.47,E2 -25938.47} C_VEL
LIN {X 0,Y 167.061,Z 417.571,A -85,B 0,C 180,E1 -25940.308,E2 -25940.308} C_VEL
LIN {X 0,Y 168.155,Z 426.384,A -85,B 0,C 180,E1 -25944.705,E2 -25944.705} C_VEL
LIN {X 0,Y 168.883,Z 436.338,A -85,B 0,C 180,E1 -25949.085,E2 -25949.085} C_VEL
LIN {X 0,Y 168.201,Z 439.052,A -85,B 0,C 180,E1 -25949.789,E2 -25949.789} C_VEL
LIN {X 0,Y 163.593,Z 450.968,A -85,B 0,C 180,E1 -25952.532,E2 -25952.532} C_VEL
LIN {X 0,Y 158.701,Z 461.579,A -85,B 0,C 180,E1 -25955.322,E2 -25955.322} C_VEL
LIN {X 0,Y 151.593,Z 472.112,A -85,B 0,C 180,E1 -25957.989,E2 -25957.989} C_VEL
LIN {X 0,Y 144.429,Z 481.509,A -85,B 0,C 180,E1 -25961.042,E2 -25961.042} C_VEL
LIN {X 0,Y 136.914,Z 490.768,A -85,B 0,C 180,E1 -25965.106,E2 -25965.106} C_VEL
LIN {X 0,Y 130.191,Z 498.483,A -85,B 0,C 180,E1 -25969.626,E2 -25969.626} C_VEL
LIN {X 0,Y 123.734,Z 505.736,A -85,B 0,C 180,E1 -25975.39,E2 -25975.39} C_VEL
LIN {X 0,Y 118.649,Z 511.479,A -85,B 0,C 180,E1 -25981.715,E2 -25981.715} C_VEL
LIN {X 0,Y 115.093,Z 515.86,A -85,B 0,C 180,E1 -25988.508,E2 -25988.508} C_VEL
LIN {X 0,Y 113.169,Z 518.988,A -85,B 0,C 180,E1 -25995.618,E2 -25995.618} C_VEL
LIN {X 0,Y 112.888,Z 520.927,A -85,B 0,C 180,E1 -26002.848,E2 -26002.848} C_VEL
LIN {X 0,Y 113.183,Z 521.447,A -85,B 0,C 180,E1 -26006.441,E2 -26006.441} C_VEL
LIN {X 0,Y 113.474,Z 521.641,A -85,B 0,C 180,E1 -26010.001,E2 -26010.001} C_VEL
LIN {X 0,Y 113.015,Z 521.137,A -85,B 0,C 180,E1 -26015.748,E2 -26015.748} C_VEL
LIN {X 0,Y 112.846,Z 520.083,A -85,B 0,C 180,E1 -26020.769,E2 -26020.769} C_VEL
LIN {X 0,Y 113.919,Z 517.531,A -85,B 0,C 180,E1 -26027.968,E2 -26027.968} C_VEL
LIN {X 0,Y 116.678,Z 513.76,A -85,B 0,C 180,E1 -26034.939,E2 -26034.939} C_VEL
LIN {X 0,Y 121.012,Z 508.687,A -85,B 0,C 180,E1 -26041.514,E2 -26041.514} C_VEL
LIN {X 0,Y 126.898,Z 502.2,A -85,B 0,C 180,E1 -26047.534,E2 -26047.534} C_VEL
LIN {X 0,Y 132.86,Z 495.441,A -85,B 0,C 180,E1 -26052.22,E2 -26052.22} C_VEL
LIN {X 0,Y 140.486,Z 486.895,A -85,B 0,C 180,E1 -26056.502,E2 -26056.502} C_VEL
LIN {X 0,Y 143.448,Z 483.708,A -85,B 0,C 180,E1 -26057.82,E2 -26057.82} C_VEL
LIN {X 0,Y 152.377,Z 482.287,A -85,B 0,C 180,E1 -26061.637,E2 -26061.637} C_VEL
LIN {X 0,Y 150.888,Z 481.626,A -85,B 0,C 180,E1 -26062.735,E2 -26062.735} C_VEL
LIN {X 0,Y 141.745,Z 478.447,A -85,B 0,C 180,E1 -26066.948,E2 -26066.948} C_VEL
LIN {X 0,Y 133.638,Z 474.254,A -85,B 0,C 180,E1 -26071.751,E2 -26071.751} C_VEL
LIN {X 0,Y 130.85,Z 472.327,A -85,B 0,C 180,E1 -26073.805,E2 -26073.805} C_VEL
LIN {X 0,Y 128.571,Z 471.682,A -85,B 0,C 180,E1 -26075.211,E2 -26075.211} C_VEL
LIN {X 0,Y 123.992,Z 472.53,A -85,B 0,C 180,E1 -26077.455,E2 -26077.455} C_VEL
LIN {X 0,Y 119.877,Z 473.612,A -85,B 0,C 180,E1 -26079.958,E2 -26079.958} C_VEL
LIN {X 0,Y 118.383,Z 473.426,A -85,B 0,C 180,E1 -26081.742,E2 -26081.742} C_VEL
LIN {X 0,Y 115.659,Z 470.967,A -85,B 0,C 180,E1 -26089.497,E2 -26089.497} C_VEL
LIN {X 0,Y 115.997,Z 467.1,A -85,B 0,C 180,E1 -26100,E2 -26100} C_VEL
LIN {X 0,Y 120.71,Z 462.672,A -85,B 0,C 180,E1 -26110.06,E2 -26110.06} C_VEL
LIN {X 0,Y 126.08,Z 459.316,A -85,B 0,C 180,E1 -26116.184,E2 -26116.184} C_VEL
LIN {X 0,Y 135.129,Z 454.458,A -85,B 0,C 180,E1 -26122.959,E2 -26122.959} C_VEL
LIN {X 0,Y 141.779,Z 450.939,A -85,B 0,C 180,E1 -26126.496,E2 -26126.496} C_VEL
LIN {X 0,Y 148.007,Z 447.835,A -85,B 0,C 180,E1 -26129.368,E2 -26129.368} C_VEL
LIN {X 0,Y 151.643,Z 445.812,A -85,B 0,C 180,E1 -26130.651,E2 -26130.651} C_VEL
LIN {X 0,Y 158.001,Z 442.616,A -85,B 0,C 180,E1 -26133,E2 -26133} C_VEL
LIN {X 0,Y 160.635,Z 441.109,A -85,B 0,C 180,E1 -26133.769,E2 -26133.769} C_VEL
LIN {X 0,Y 161.327,Z 441.003,A -85,B 0,C 180,E1 -26134.135,E2 -26134.135} C_VEL
LIN {X 0,Y 155.071,Z 450.766,A -85,B 0,C 180,E1 -26136.442,E2 -26136.442} C_VEL
LIN {X 0,Y 147.992,Z 460.683,A -85,B 0,C 180,E1 -26139.492,E2 -26139.492} C_VEL
LIN {X 0,Y 140.009,Z 470.366,A -85,B 0,C 180,E1 -26143.292,E2 -26143.292} C_VEL
LIN {X 0,Y 132.686,Z 478.38,A -85,B 0,C 180,E1 -26147.52,E2 -26147.52} C_VEL
LIN {X 0,Y 126.176,Z 484.978,A -85,B 0,C 180,E1 -26152.214,E2 -26152.214} C_VEL
LIN {X 0,Y 119.634,Z 491.078,A -85,B 0,C 180,E1 -26158.081,E2 -26158.081} C_VEL
LIN {X 0,Y 114.393,Z 495.771,A -85,B 0,C 180,E1 -26164.528,E2 -26164.528} C_VEL
LIN {X 0,Y 110.446,Z 499.197,A -85,B 0,C 180,E1 -26171.447,E2 -26171.447} C_VEL
LIN {X 0,Y 107.908,Z 501.439,A -85,B 0,C 180,E1 -26178.732,E2 -26178.732} C_VEL
LIN {X 0,Y 106.733,Z 502.564,A -85,B 0,C 180,E1 -26186.224,E2 -26186.224} C_VEL
LIN {X 0,Y 106.72,Z 502.574,A -85,B 0,C 180,E1 -26193.775,E2 -26193.775} C_VEL
LIN {X 0,Y 107.904,Z 501.48,A -85,B 0,C 180,E1 -26201.267,E2 -26201.267} C_VEL
LIN {X 0,Y 110.443,Z 499.274,A -85,B 0,C 180,E1 -26208.552,E2 -26208.552} C_VEL
LIN {X 0,Y 114.346,Z 495.897,A -85,B 0,C 180,E1 -26215.482,E2 -26215.482} C_VEL
LIN {X 0,Y 119.569,Z 491.249,A -85,B 0,C 180,E1 -26221.937,E2 -26221.937} C_VEL
LIN {X 0,Y 126.091,Z 485.186,A -85,B 0,C 180,E1 -26227.814,E2 -26227.814} C_VEL
LIN {X 0,Y 133.607,Z 477.548,A -85,B 0,C 180,E1 -26233.143,E2 -26233.143} C_VEL
LIN {X 0,Y 141.029,Z 469.368,A -85,B 0,C 180,E1 -26237.31,E2 -26237.31} C_VEL
LIN {X 0,Y 147.894,Z 461.038,A -85,B 0,C 180,E1 -26240.552,E2 -26240.552} C_VEL
LIN {X 0,Y 154.889,Z 451.287,A -85,B 0,C 180,E1 -26243.578,E2 -26243.578} C_VEL
LIN {X 0,Y 162.204,Z 440.01,A -85,B 0,C 180,E1 -26246.191,E2 -26246.191} C_VEL
LIN {X 0,Y 162.803,Z 438.569,A -85,B 0,C 180,E1 -26246.667,E2 -26246.667} C_VEL
LIN {X 0,Y 163.354,Z 433.892,A -85,B 0,C 180,E1 -26248.917,E2 -26248.917} C_VEL
LIN {X 0,Y 163.266,Z 428.925,A -85,B 0,C 180,E1 -26251.737,E2 -26251.737} C_VEL
LIN {X 0,Y 162.544,Z 422.966,A -85,B 0,C 180,E1 -26255.746,E2 -26255.746} C_VEL
LIN {X 0,Y 161.782,Z 419.091,A -85,B 0,C 180,E1 -26258.842,E2 -26258.842} C_VEL
LIN {X 0,Y 160.631,Z 414.236,A -85,B 0,C 180,E1 -26263.608,E2 -26263.608} C_VEL
LIN {X 0,Y 159.814,Z 411.514,A -85,B 0,C 180,E1 -26267.298,E2 -26267.298} C_VEL
LIN {X 0,Y 159.41,Z 410.008,A -85,B 0,C 180,E1 -26269.842,E2 -26269.842} C_VEL
LIN {X 0,Y 159.03,Z 408.999,A -85,B 0,C 180,E1 -26272.381,E2 -26272.381} C_VEL
LIN {X 0,Y 159.049,Z 407.558,A -85,B 0,C 180,E1 -26280,E2 -26280} C_VEL
LIN {X 0,Y 159.262,Z 409.614,A -85,B 0,C 180,E1 -26285.063,E2 -26285.063} C_VEL
LIN {X 0,Y 160.179,Z 412.87,A -85,B 0,C 180,E1 -26290.108,E2 -26290.108} C_VEL
LIN {X 0,Y 160.947,Z 414.843,A -85,B 0,C 180,E1 -26292.611,E2 -26292.611} C_VEL
LIN {X 0,Y 162.655,Z 420.168,A -85,B 0,C 180,E1 -26297.605,E2 -26297.605} C_VEL
LIN {X 0,Y 163.146,Z 423.081,A -85,B 0,C 180,E1 -26299.502,E2 -26299.502} C_VEL
LIN {X 0,Y 163.768,Z 431.838,A -85,B 0,C 180,E1 -26304.059,E2 -26304.059} C_VEL
LIN {X 0,Y 163.949,Z 439.947,A -85,B 0,C 180,E1 -26307.786,E2 -26307.786} C_VEL
LIN {X 0,Y 159.131,Z 451.534,A -85,B 0,C 180,E1 -26310.547,E2 -26310.547} C_VEL
LIN {X 0,Y 153.917,Z 462.094,A -85,B 0,C 180,E1 -26313.41,E2 -26313.41} C_VEL
LIN {X 0,Y 146.027,Z 473.144,A -85,B 0,C 180,E1 -26316.28,E2 -26316.28} C_VEL
LIN {X 0,Y 138.65,Z 482.312,A -85,B 0,C 180,E1 -26319.377,E2 -26319.377} C_VEL
LIN {X 0,Y 130.838,Z 491.345,A -85,B 0,C 180,E1 -26323.519,E2 -26323.519} C_VEL
LIN {X 0,Y 122.949,Z 499.837,A -85,B 0,C 180,E1 -26328.902,E2 -26328.902} C_VEL
LIN {X 0,Y 116.364,Z 506.696,A -85,B 0,C 180,E1 -26334.987,E2 -26334.987} C_VEL
LIN {X 0,Y 111.094,Z 512.209,A -85,B 0,C 180,E1 -26341.882,E2 -26341.882} C_VEL
LIN {X 0,Y 108.418,Z 515.242,A -85,B 0,C 180,E1 -26347.112,E2 -26347.112} C_VEL
LIN {X 0,Y 106.228,Z 518.371,A -85,B 0,C 180,E1 -26354.655,E2 -26354.655} C_VEL
LIN {X 0,Y 105.779,Z 520.311,A -85,B 0,C 180,E1 -26362.365,E2 -26362.365} C_VEL
LIN {X 0,Y 106.076,Z 520.835,A -85,B 0,C 180,E1 -26366.202,E2 -26366.202} C_VEL
LIN {X 0,Y 106.386,Z 521.031,A -85,B 0,C 180,E1 -26370.001,E2 -26370.001} C_VEL
LIN {X 0,Y 105.942,Z 520.587,A -85,B 0,C 180,E1 -26375.692,E2 -26375.692} C_VEL
LIN {X 0,Y 105.794,Z 519.465,A -85,B 0,C 180,E1 -26381.496,E2 -26381.496} C_VEL
LIN {X 0,Y 107.103,Z 516.913,A -85,B 0,C 180,E1 -26389.154,E2 -26389.154} C_VEL
LIN {X 0,Y 110.47,Z 512.812,A -85,B 0,C 180,E1 -26397.043,E2 -26397.043} C_VEL
LIN {X 0,Y 114.943,Z 508.068,A -85,B 0,C 180,E1 -26403.388,E2 -26403.388} C_VEL
LIN {X 0,Y 121.258,Z 501.58,A -85,B 0,C 180,E1 -26409.61,E2 -26409.61} C_VEL
LIN {X 0,Y 127.147,Z 495.347,A -85,B 0,C 180,E1 -26414.064,E2 -26414.064} C_VEL
LIN {X 0,Y 134.487,Z 487.532,A -85,B 0,C 180,E1 -26418.132,E2 -26418.132} C_VEL
LIN {X 0,Y 139.745,Z 481.9,A -85,B 0,C 180,E1 -26420.363,E2 -26420.363} C_VEL
LIN {X 0,Y 143.065,Z 481.525,A -85,B 0,C 180,E1 -26421.814,E2 -26421.814} C_VEL
LIN {X 0,Y 135.846,Z 478.604,A -85,B 0,C 180,E1 -26425.314,E2 -26425.314} C_VEL
LIN {X 0,Y 133.093,Z 477.401,A -85,B 0,C 180,E1 -26426.781,E2 -26426.781} C_VEL
LIN {X 0,Y 127.844,Z 476.777,A -85,B 0,C 180,E1 -26430.347,E2 -26430.347} C_VEL
LIN {X 0,Y 119.602,Z 474.282,A -85,B 0,C 180,E1 -26439.356,E2 -26439.356} C_VEL
LIN {X 0,Y 118.383,Z 473.426,A -85,B 0,C 180,E1 -26441.742,E2 -26441.742} C_VEL
LIN {X 0,Y 116.696,Z 472.903,A -85,B 0,C 180,E1 -26444.488,E2 -26444.488} C_VEL
LIN {X 0,Y 113.072,Z 473.251,A -85,B 0,C 180,E1 -26449.094,E2 -26449.094} C_VEL
LIN {X 0,Y 110.293,Z 473.541,A -85,B 0,C 180,E1 -26453.967,E2 -26453.967} C_VEL
LIN {X 0,Y 109.958,Z 472.934,A -85,B 0,C 180,E1 -26457.007,E2 -26457.007} C_VEL
LIN {X 0,Y 115.362,Z 467.61,A -85,B 0,C 180,E1 -26470.531,E2 -26470.531} C_VEL
LIN {X 0,Y 124.397,Z 462.542,A -85,B 0,C 180,E1 -26479.815,E2 -26479.815} C_VEL
LIN {X 0,Y 132.423,Z 458.703,A -85,B 0,C 180,E1 -26485.124,E2 -26485.124} C_VEL
LIN {X 0,Y 144.306,Z 453.073,A -85,B 0,C 180,E1 -26490.756,E2 -26490.756} C_VEL
LIN {X 0,Y 152.403,Z 449.081,A -85,B 0,C 180,E1 -26493.599,E2 -26493.599} C_VEL
LIN {X 0,Y 151.547,Z 450.588,A -85,B 0,C 180,E1 -26494.079,E2 -26494.079} C_VEL
LIN {X 0,Y 143.596,Z 461.289,A -85,B 0,C 180,E1 -26497.313,E2 -26497.313} C_VEL
LIN {X 0,Y 135.258,Z 470.973,A -85,B 0,C 180,E1 -26501.112,E2 -26501.112} C_VEL
LIN {X 0,Y 127.543,Z 478.989,A -85,B 0,C 180,E1 -26505.367,E2 -26505.367} C_VEL
LIN {X 0,Y 120.647,Z 485.587,A -85,B 0,C 180,E1 -26510.149,E2 -26510.149} C_VEL
LIN {X 0,Y 113.665,Z 491.69,A -85,B 0,C 180,E1 -26516.186,E2 -26516.186} C_VEL
LIN {X 0,Y 108.027,Z 496.381,A -85,B 0,C 180,E1 -26522.908,E2 -26522.908} C_VEL
LIN {X 0,Y 103.767,Z 499.805,A -85,B 0,C 180,E1 -26530.205,E2 -26530.205} C_VEL
LIN {X 0,Y 100.991,Z 502.047,A -85,B 0,C 180,E1 -26537.949,E2 -26537.949} C_VEL
LIN {X 0,Y 99.672,Z 503.173,A -85,B 0,C 180,E1 -26545.956,E2 -26545.956} C_VEL
LIN {X 0,Y 99.659,Z 503.182,A -85,B 0,C 180,E1 -26554.043,E2 -26554.043} C_VEL
LIN {X 0,Y 100.987,Z 502.087,A -85,B 0,C 180,E1 -26562.05,E2 -26562.05} C_VEL
LIN {X 0,Y 103.764,Z 499.882,A -85,B 0,C 180,E1 -26569.794,E2 -26569.794} C_VEL
LIN {X 0,Y 107.979,Z 496.506,A -85,B 0,C 180,E1 -26577.103,E2 -26577.103} C_VEL
LIN {X 0,Y 113.6,Z 491.858,A -85,B 0,C 180,E1 -26583.833,E2 -26583.833} C_VEL
LIN {X 0,Y 120.561,Z 485.793,A -85,B 0,C 180,E1 -26589.883,E2 -26589.883} C_VEL
LIN {X 0,Y 128.529,Z 478.153,A -85,B 0,C 180,E1 -26595.303,E2 -26595.303} C_VEL
LIN {X 0,Y 136.338,Z 469.969,A -85,B 0,C 180,E1 -26599.493,E2 -26599.493} C_VEL
LIN {X 0,Y 143.5,Z 461.64,A -85,B 0,C 180,E1 -26602.735,E2 -26602.735} C_VEL
LIN {X 0,Y 150.759,Z 451.939,A -85,B 0,C 180,E1 -26605.727,E2 -26605.727} C_VEL
LIN {X 0,Y 157.446,Z 442.082,A -85,B 0,C 180,E1 -26608.006,E2 -26608.006} C_VEL
LIN {X 0,Y 157.954,Z 440.76,A -85,B 0,C 180,E1 -26608.511,E2 -26608.511} C_VEL
LIN {X 0,Y 158.478,Z 436.536,A -85,B 0,C 180,E1 -26610.803,E2 -26610.803} C_VEL
LIN {X 0,Y 158.483,Z 432.06,A -85,B 0,C 180,E1 -26613.675,E2 -26613.675} C_VEL
LIN {X 0,Y 158.062,Z 426.529,A -85,B 0,C 180,E1 -26617.793,E2 -26617.793} C_VEL
LIN {X 0,Y 157.391,Z 422.286,A -85,B 0,C 180,E1 -26621.785,E2 -26621.785} C_VEL
LIN {X 0,Y 156.944,Z 419.909,A -85,B 0,C 180,E1 -26624.414,E2 -26624.414} C_VEL
LIN {X 0,Y 156.203,Z 416.544,A -85,B 0,C 180,E1 -26629.632,E2 -26629.632} C_VEL
LIN {X 0,Y 155.885,Z 415.32,A -85,B 0,C 180,E1 -26632.68,E2 -26632.68} C_VEL
LIN {X 0,Y 156.084,Z 414.044,A -85,B 0,C 180,E1 -26640,E2 -26640} C_VEL
LIN {X 0,Y 156.207,Z 416.214,A -85,B 0,C 180,E1 -26645.162,E2 -26645.162} C_VEL
LIN {X 0,Y 157.35,Z 420.503,A -85,B 0,C 180,E1 -26651.595,E2 -26651.595} C_VEL
LIN {X 0,Y 158.781,Z 425.592,A -85,B 0,C 180,E1 -26656.72,E2 -26656.72} C_VEL
LIN {X 0,Y 159.09,Z 428.686,A -85,B 0,C 180,E1 -26658.813,E2 -26658.813} C_VEL
LIN {X 0,Y 159.193,Z 437.177,A -85,B 0,C 180,E1 -26663.411,E2 -26663.411} C_VEL
LIN {X 0,Y 159.054,Z 442.891,A -85,B 0,C 180,E1 -26666.222,E2 -26666.222} C_VEL
LIN {X 0,Y 153.181,Z 455.431,A -85,B 0,C 180,E1 -26669.341,E2 -26669.341} C_VEL
LIN {X 0,Y 148.573,Z 463.697,A -85,B 0,C 180,E1 -26671.63,E2 -26671.63} C_VEL
LIN {X 0,Y 140.598,Z 474.174,A -85,B 0,C 180,E1 -26674.435,E2 -26674.435} C_VEL
LIN {X 0,Y 132.989,Z 483.071,A -85,B 0,C 180,E1 -26677.563,E2 -26677.563} C_VEL
LIN {X 0,Y 124.892,Z 491.869,A -85,B 0,C 180,E1 -26681.789,E2 -26681.789} C_VEL
LIN {X 0,Y 117.605,Z 499.22,A -85,B 0,C 180,E1 -26686.59,E2 -26686.59} C_VEL
LIN {X 0,Y 110.529,Z 506.077,A -85,B 0,C 180,E1 -26692.84,E2 -26692.84} C_VEL
LIN {X 0,Y 104.921,Z 511.48,A -85,B 0,C 180,E1 -26699.844,E2 -26699.844} C_VEL
LIN {X 0,Y 101.824,Z 514.624,A -85,B 0,C 180,E1 -26705.537,E2 -26705.537} C_VEL
LIN {X 0,Y 99.311,Z 517.753,A -85,B 0,C 180,E1 -26713.557,E2 -26713.557} C_VEL
LIN {X 0,Y 98.692,Z 519.695,A -85,B 0,C 180,E1 -26721.813,E2 -26721.813} C_VEL
LIN {X 0,Y 98.973,Z 520.222,A -85,B 0,C 180,E1 -26725.929,E2 -26725.929} C_VEL
LIN {X 0,Y 99.299,Z 520.422,A -85,B 0,C 180,E1 -26730.001,E2 -26730.001} C_VEL
LIN {X 0,Y 98.87,Z 520.036,A -85,B 0,C 180,E1 -26735.64,E2 -26735.64} C_VEL
LIN {X 0,Y 98.782,Z 518.848,A -85,B 0,C 180,E1 -26742.325,E2 -26742.325} C_VEL
LIN {X 0,Y 100.345,Z 516.295,A -85,B 0,C 180,E1 -26750.5,E2 -26750.5} C_VEL
LIN {X 0,Y 103.767,Z 512.518,A -85,B 0,C 180,E1 -26758.302,E2 -26758.302} C_VEL
LIN {X 0,Y 108.987,Z 507.447,A -85,B 0,C 180,E1 -26765.477,E2 -26765.477} C_VEL
LIN {X 0,Y 115.783,Z 500.958,A -85,B 0,C 180,E1 -26771.891,E2 -26771.891} C_VEL
LIN {X 0,Y 122.124,Z 494.709,A -85,B 0,C 180,E1 -26776.417,E2 -26776.417} C_VEL
LIN {X 0,Y 129.845,Z 486.921,A -85,B 0,C 180,E1 -26780.471,E2 -26780.471} C_VEL
LIN {X 0,Y 133.682,Z 482.969,A -85,B 0,C 180,E1 -26782.055,E2 -26782.055} C_VEL
LIN {X 0,Y 126.897,Z 481.766,A -85,B 0,C 180,E1 -26786.37,E2 -26786.37} C_VEL
LIN {X 0,Y 123.065,Z 481.234,A -85,B 0,C 180,E1 -26789.072,E2 -26789.072} C_VEL
LIN {X 0,Y 114.456,Z 478.785,A -85,B 0,C 180,E1 -26798.382,E2 -26798.382} C_VEL
LIN {X 0,Y 109.877,Z 473.176,A -85,B 0,C 180,E1 -26816.333,E2 -26816.333} C_VEL
LIN {X 0,Y 109.958,Z 472.934,A -85,B 0,C 180,E1 -26817.007,E2 -26817.007} C_VEL
LIN {X 0,Y 110.011,Z 472.264,A -85,B 0,C 180,E1 -26820.065,E2 -26820.065} C_VEL
LIN {X 0,Y 109.695,Z 472.231,A -85,B 0,C 180,E1 -26829.374,E2 -26829.374} C_VEL
LIN {X 0,Y 110.863,Z 471.676,A -85,B 0,C 180,E1 -26832.357,E2 -26832.357} C_VEL
LIN {X 0,Y 111.52,Z 471.308,A -85,B 0,C 180,E1 -26833.292,E2 -26833.292} C_VEL
LIN {X 0,Y 121.915,Z 466.194,A -85,B 0,C 180,E1 -26842.726,E2 -26842.726} C_VEL
LIN {X 0,Y 129.743,Z 462.746,A -85,B 0,C 180,E1 -26847.415,E2 -26847.415} C_VEL
LIN {X 0,Y 142.324,Z 457.275,A -85,B 0,C 180,E1 -26852.901,E2 -26852.901} C_VEL
LIN {X 0,Y 143.21,Z 457.151,A -85,B 0,C 180,E1 -26853.458,E2 -26853.458} C_VEL
LIN {X 0,Y 135.661,Z 466.247,A -85,B 0,C 180,E1 -26856.582,E2 -26856.582} C_VEL
LIN {X 0,Y 127.169,Z 475.181,A -85,B 0,C 180,E1 -26860.544,E2 -26860.544} C_VEL
LIN {X 0,Y 119.305,Z 482.578,A -85,B 0,C 180,E1 -26865.016,E2 -26865.016} C_VEL
LIN {X 0,Y 113.33,Z 487.873,A -85,B 0,C 180,E1 -26869.371,E2 -26869.371} C_VEL
LIN {X 0,Y 106.206,Z 493.615,A -85,B 0,C 180,E1 -26875.772,E2 -26875.772} C_VEL
LIN {X 0,Y 101.762,Z 496.992,A -85,B 0,C 180,E1 -26881.089,E2 -26881.089} C_VEL
LIN {X 0,Y 97.124,Z 500.415,A -85,B 0,C 180,E1 -26888.788,E2 -26888.788} C_VEL
LIN {X 0,Y 94.097,Z 502.654,A -85,B 0,C 180,E1 -26897.051,E2 -26897.051} C_VEL
LIN {X 0,Y 92.615,Z 503.782,A -85,B 0,C 180,E1 -26905.647,E2 -26905.647} C_VEL
LIN {X 0,Y 92.603,Z 503.791,A -85,B 0,C 180,E1 -26914.352,E2 -26914.352} C_VEL
LIN {X 0,Y 94.094,Z 502.694,A -85,B 0,C 180,E1 -26922.948,E2 -26922.948} C_VEL
LIN {X 0,Y 97.12,Z 500.491,A -85,B 0,C 180,E1 -26931.211,E2 -26931.211} C_VEL
LIN {X 0,Y 101.718,Z 497.115,A -85,B 0,C 180,E1 -26938.923,E2 -26938.923} C_VEL
LIN {X 0,Y 107.772,Z 492.467,A -85,B 0,C 180,E1 -26945.937,E2 -26945.937} C_VEL
LIN {X 0,Y 115.208,Z 486.4,A -85,B 0,C 180,E1 -26952.146,E2 -26952.146} C_VEL
LIN {X 0,Y 123.659,Z 478.756,A -85,B 0,C 180,E1 -26957.632,E2 -26957.632} C_VEL
LIN {X 0,Y 131.847,Z 470.572,A -85,B 0,C 180,E1 -26961.834,E2 -26961.834} C_VEL
LIN {X 0,Y 139.324,Z 462.242,A -85,B 0,C 180,E1 -26965.055,E2 -26965.055} C_VEL
LIN {X 0,Y 147.426,Z 451.834,A -85,B 0,C 180,E1 -26968.198,E2 -26968.198} C_VEL
LIN {X 0,Y 152.427,Z 444.771,A -85,B 0,C 180,E1 -26969.825,E2 -26969.825} C_VEL
LIN {X 0,Y 153.226,Z 442.779,A -85,B 0,C 180,E1 -26970.629,E2 -26970.629} C_VEL
LIN {X 0,Y 153.733,Z 438.232,A -85,B 0,C 180,E1 -26973.53,E2 -26973.53} C_VEL
LIN {X 0,Y 153.777,Z 433.448,A -85,B 0,C 180,E1 -26977.139,E2 -26977.139} C_VEL
LIN {X 0,Y 153.615,Z 430.731,A -85,B 0,C 180,E1 -26979.531,E2 -26979.531} C_VEL
LIN {X 0,Y 153.161,Z 426.095,A -85,B 0,C 180,E1 -26984.495,E2 -26984.495} C_VEL
LIN {X 0,Y 152.718,Z 422.964,A -85,B 0,C 180,E1 -26989.392,E2 -26989.392} C_VEL
LIN {X 0,Y 152.533,Z 421.841,A -85,B 0,C 180,E1 -26992.054,E2 -26992.054} C_VEL
LIN {X 0,Y 152.545,Z 420.668,A -85,B 0,C 180,E1 -26997.359,E2 -26997.359} C_VEL
LIN {X 0,Y 152.85,Z 420.417,A -85,B 0,C 180,E1 -27000,E2 -27000} C_VEL
LIN {X 0,Y 152.88,Z 422.683,A -85,B 0,C 180,E1 -27005.275,E2 -27005.275} C_VEL
LIN {X 0,Y 153.595,Z 426.037,A -85,B 0,C 180,E1 -27010.546,E2 -27010.546} C_VEL
LIN {X 0,Y 154.743,Z 430.924,A -85,B 0,C 180,E1 -27015.813,E2 -27015.813} C_VEL
LIN {X 0,Y 154.874,Z 433.411,A -85,B 0,C 180,E1 -27017.647,E2 -27017.647} C_VEL
LIN {X 0,Y 154.555,Z 440.663,A -85,B 0,C 180,E1 -27021.823,E2 -27021.823} C_VEL
LIN {X 0,Y 154.24,Z 445.412,A -85,B 0,C 180,E1 -27024.315,E2 -27024.315} C_VEL
LIN {X 0,Y 152.675,Z 448.95,A -85,B 0,C 180,E1 -27025.319,E2 -27025.319} C_VEL
LIN {X 0,Y 145.951,Z 461.286,A -85,B 0,C 180,E1 -27028.649,E2 -27028.649} C_VEL
LIN {X 0,Y 143.553,Z 464.971,A -85,B 0,C 180,E1 -27029.659,E2 -27029.659} C_VEL
LIN {X 0,Y 135.329,Z 475.189,A -85,B 0,C 180,E1 -27032.446,E2 -27032.446} C_VEL
LIN {X 0,Y 126.247,Z 485.182,A -85,B 0,C 180,E1 -27036.178,E2 -27036.178} C_VEL
LIN {X 0,Y 117.951,Z 493.515,A -85,B 0,C 180,E1 -27040.549,E2 -27040.549} C_VEL
LIN {X 0,Y 110.443,Z 500.458,A -85,B 0,C 180,E1 -27045.576,E2 -27045.576} C_VEL
LIN {X 0,Y 103.196,Z 506.933,A -85,B 0,C 180,E1 -27052.2,E2 -27052.2} C_VEL
LIN {X 0,Y 97.049,Z 512.344,A -85,B 0,C 180,E1 -27060.342,E2 -27060.342} C_VEL
LIN {X 0,Y 93.614,Z 515.721,A -85,B 0,C 180,E1 -27067.954,E2 -27067.954} C_VEL
LIN {X 0,Y 91.766,Z 518.253,A -85,B 0,C 180,E1 -27076.718,E2 -27076.718} C_VEL
LIN {X 0,Y 91.889,Z 519.611,A -85,B 0,C 180,E1 -27085.615,E2 -27085.615} C_VEL
LIN {X 0,Y 92.211,Z 519.812,A -85,B 0,C 180,E1 -27090.001,E2 -27090.001} C_VEL
LIN {X 0,Y 91.802,Z 519.482,A -85,B 0,C 180,E1 -27095.606,E2 -27095.606} C_VEL
LIN {X 0,Y 91.772,Z 518.23,A -85,B 0,C 180,E1 -27103.283,E2 -27103.283} C_VEL
LIN {X 0,Y 93.628,Z 515.674,A -85,B 0,C 180,E1 -27112.045,E2 -27112.045} C_VEL
LIN {X 0,Y 97.476,Z 511.897,A -85,B 0,C 180,E1 -27120.312,E2 -27120.312} C_VEL
LIN {X 0,Y 103.206,Z 506.827,A -85,B 0,C 180,E1 -27127.799,E2 -27127.799} C_VEL
LIN {X 0,Y 110.512,Z 500.338,A -85,B 0,C 180,E1 -27134.392,E2 -27134.392} C_VEL
LIN {X 0,Y 118.156,Z 493.288,A -85,B 0,C 180,E1 -27139.435,E2 -27139.435} C_VEL
LIN {X 0,Y 124.14,Z 487.549,A -85,B 0,C 180,E1 -27142.429,E2 -27142.429} C_VEL
LIN {X 0,Y 124.825,Z 486.368,A -85,B 0,C 180,E1 -27143.216,E2 -27143.216} C_VEL
LIN {X 0,Y 118.205,Z 485.461,A -85,B 0,C 180,E1 -27147.649,E2 -27147.649} C_VEL
LIN {X 0,Y 109.182,Z 483.059,A -85,B 0,C 180,E1 -27157.281,E2 -27157.281} C_VEL
LIN {X 0,Y 104.219,Z 478.776,A -85,B 0,C 180,E1 -27172.249,E2 -27172.249} C_VEL
LIN {X 0,Y 107.644,Z 473.723,A -85,B 0,C 180,E1 -27187.503,E2 -27187.503} C_VEL
LIN {X 0,Y 111.52,Z 471.308,A -85,B 0,C 180,E1 -27193.292,E2 -27193.292} C_VEL
LIN {X 0,Y 113.415,Z 470.463,A -85,B 0,C 180,E1 -27196.115,E2 -27196.115} C_VEL
LIN {X 0,Y 118.722,Z 469.726,A -85,B 0,C 180,E1 -27204.518,E2 -27204.518} C_VEL
LIN {X 0,Y 121.615,Z 468.873,A -85,B 0,C 180,E1 -27206.917,E2 -27206.917} C_VEL
LIN {X 0,Y 122.794,Z 468.406,A -85,B 0,C 180,E1 -27207.615,E2 -27207.615} C_VEL
LIN {X 0,Y 133.417,Z 464.079,A -85,B 0,C 180,E1 -27212.558,E2 -27212.558} C_VEL
LIN {X 0,Y 134.176,Z 463.959,A -85,B 0,C 180,E1 -27213.063,E2 -27213.063} C_VEL
LIN {X 0,Y 125.149,Z 473.392,A -85,B 0,C 180,E1 -27216.846,E2 -27216.846} C_VEL
LIN {X 0,Y 116.715,Z 481.226,A -85,B 0,C 180,E1 -27221.175,E2 -27221.175} C_VEL
LIN {X 0,Y 110.114,Z 486.809,A -85,B 0,C 180,E1 -27225.405,E2 -27225.405} C_VEL
LIN {X 0,Y 102.165,Z 492.912,A -85,B 0,C 180,E1 -27231.747,E2 -27231.747} C_VEL
LIN {X 0,Y 95.619,Z 497.602,A -85,B 0,C 180,E1 -27239.035,E2 -27239.035} C_VEL
LIN {X 0,Y 90.564,Z 501.024,A -85,B 0,C 180,E1 -27247.168,E2 -27247.168} C_VEL
LIN {X 0,Y 87.231,Z 503.262,A -85,B 0,C 180,E1 -27256.012,E2 -27256.012} C_VEL
LIN {X 0,Y 85.564,Z 504.39,A -85,B 0,C 180,E1 -27265.288,E2 -27265.288} C_VEL
LIN {X 0,Y 85.552,Z 504.399,A -85,B 0,C 180,E1 -27274.711,E2 -27274.711} C_VEL
LIN {X 0,Y 87.228,Z 503.301,A -85,B 0,C 180,E1 -27283.987,E2 -27283.987} C_VEL
LIN {X 0,Y 90.56,Z 501.099,A -85,B 0,C 180,E1 -27292.831,E2 -27292.831} C_VEL
LIN {X 0,Y 95.576,Z 497.723,A -85,B 0,C 180,E1 -27300.978,E2 -27300.978} C_VEL
LIN {X 0,Y 102.107,Z 493.075,A -85,B 0,C 180,E1 -27308.276,E2 -27308.276} C_VEL
LIN {X 0,Y 110.055,Z 487.007,A -85,B 0,C 180,E1 -27314.623,E2 -27314.623} C_VEL
LIN {X 0,Y 117.813,Z 480.446,A -85,B 0,C 180,E1 -27319.515,E2 -27319.515} C_VEL
LIN {X 0,Y 126.327,Z 472.466,A -85,B 0,C 180,E1 -27323.772,E2 -27323.772} C_VEL
LIN {X 0,Y 135.386,Z 462.844,A -85,B 0,C 180,E1 -27327.516,E2 -27327.516} C_VEL
LIN {X 0,Y 143.574,Z 452.742,A -85,B 0,C 180,E1 -27330.516,E2 -27330.516} C_VEL
LIN {X 0,Y 147.588,Z 447.354,A -85,B 0,C 180,E1 -27331.753,E2 -27331.753} C_VEL
LIN {X 0,Y 148.398,Z 445.734,A -85,B 0,C 180,E1 -27332.411,E2 -27332.411} C_VEL
LIN {X 0,Y 148.92,Z 442.23,A -85,B 0,C 180,E1 -27334.866,E2 -27334.866} C_VEL
LIN {X 0,Y 149.185,Z 438.514,A -85,B 0,C 180,E1 -27337.859,E2 -27337.859} C_VEL
LIN {X 0,Y 149.236,Z 435.498,A -85,B 0,C 180,E1 -27340.752,E2 -27340.752} C_VEL
LIN {X 0,Y 149.146,Z 431.837,A -85,B 0,C 180,E1 -27344.927,E2 -27344.927} C_VEL
LIN {X 0,Y 148.945,Z 429.277,A -85,B 0,C 180,E1 -27349.12,E2 -27349.12} C_VEL
LIN {X 0,Y 148.891,Z 427.866,A -85,B 0,C 180,E1 -27352.41,E2 -27352.41} C_VEL
LIN {X 0,Y 149.027,Z 426.873,A -85,B 0,C 180,E1 -27357.297,E2 -27357.297} C_VEL
LIN {X 0,Y 149.337,Z 426.662,A -85,B 0,C 180,E1 -27360,E2 -27360} C_VEL
LIN {X 0,Y 149.296,Z 428.994,A -85,B 0,C 180,E1 -27365.402,E2 -27365.402} C_VEL
LIN {X 0,Y 149.867,Z 432.453,A -85,B 0,C 180,E1 -27370.811,E2 -27370.811} C_VEL
LIN {X 0,Y 150.518,Z 436.118,A -85,B 0,C 180,E1 -27374.88,E2 -27374.88} C_VEL
LIN {X 0,Y 150.603,Z 437.783,A -85,B 0,C 180,E1 -27376.26,E2 -27376.26} C_VEL
LIN {X 0,Y 149.716,Z 445.952,A -85,B 0,C 180,E1 -27381.215,E2 -27381.215} C_VEL
LIN {X 0,Y 149.19,Z 449.058,A -85,B 0,C 180,E1 -27382.869,E2 -27382.869} C_VEL
LIN {X 0,Y 142.638,Z 460.452,A -85,B 0,C 180,E1 -27385.947,E2 -27385.947} C_VEL
LIN {X 0,Y 139.552,Z 465.098,A -85,B 0,C 180,E1 -27387.284,E2 -27387.284} C_VEL
LIN {X 0,Y 131.628,Z 474.581,A -85,B 0,C 180,E1 -27389.817,E2 -27389.817} C_VEL
LIN {X 0,Y 122.136,Z 484.568,A -85,B 0,C 180,E1 -27393.451,E2 -27393.451} C_VEL
LIN {X 0,Y 113.375,Z 492.912,A -85,B 0,C 180,E1 -27397.784,E2 -27397.784} C_VEL
LIN {X 0,Y 105.412,Z 499.841,A -85,B 0,C 180,E1 -27402.83,E2 -27402.83} C_VEL
LIN {X 0,Y 97.593,Z 506.315,A -85,B 0,C 180,E1 -27409.601,E2 -27409.601} C_VEL
LIN {X 0,Y 90.55,Z 512.004,A -85,B 0,C 180,E1 -27418.622,E2 -27418.622} C_VEL
LIN {X 0,Y 86.983,Z 515.102,A -85,B 0,C 180,E1 -27426.174,E2 -27426.174} C_VEL
LIN {X 0,Y 84.8,Z 517.637,A -85,B 0,C 180,E1 -27435.605,E2 -27435.605} C_VEL
LIN {X 0,Y 84.784,Z 518.998,A -85,B 0,C 180,E1 -27445.246,E2 -27445.246} C_VEL
LIN {X 0,Y 85.123,Z 519.202,A -85,B 0,C 180,E1 -27450.001,E2 -27450.001} C_VEL
LIN {X 0,Y 84.72,Z 518.938,A -85,B 0,C 180,E1 -27455.463,E2 -27455.463} C_VEL
LIN {X 0,Y 84.807,Z 517.612,A -85,B 0,C 180,E1 -27464.397,E2 -27464.397} C_VEL
LIN {X 0,Y 86.999,Z 515.055,A -85,B 0,C 180,E1 -27473.824,E2 -27473.824} C_VEL
LIN {X 0,Y 91.328,Z 511.277,A -85,B 0,C 180,E1 -27482.595,E2 -27482.595} C_VEL
LIN {X 0,Y 97.606,Z 506.207,A -85,B 0,C 180,E1 -27490.395,E2 -27490.395} C_VEL
LIN {X 0,Y 105.475,Z 499.717,A -85,B 0,C 180,E1 -27497.136,E2 -27497.136} C_VEL
LIN {X 0,Y 113.51,Z 492.769,A -85,B 0,C 180,E1 -27502.131,E2 -27502.131} C_VEL
LIN {X 0,Y 114.755,Z 491.637,A -85,B 0,C 180,E1 -27502.767,E2 -27502.767} C_VEL
LIN {X 0,Y 116.002,Z 489.801,A -85,B 0,C 180,E1 -27504.181,E2 -27504.181} C_VEL
LIN {X 0,Y 109.793,Z 488.647,A -85,B 0,C 180,E1 -27509.197,E2 -27509.197} C_VEL
LIN {X 0,Y 103.79,Z 487.104,A -85,B 0,C 180,E1 -27516.029,E2 -27516.029} C_VEL
LIN {X 0,Y 98.398,Z 482.959,A -85,B 0,C 180,E1 -27531.788,E2 -27531.788} C_VEL
LIN {X 0,Y 101.894,Z 478.09,A -85,B 0,C 180,E1 -27547.93,E2 -27547.93} C_VEL
LIN {X 0,Y 110.11,Z 473.726,A -85,B 0,C 180,E1 -27558.611,E2 -27558.611} C_VEL
LIN {X 0,Y 122.794,Z 468.406,A -85,B 0,C 180,E1 -27567.615,E2 -27567.615} C_VEL
LIN {X 0,Y 123.821,Z 468.317,A -85,B 0,C 180,E1 -27568.639,E2 -27568.639} C_VEL
LIN {X 0,Y 123.958,Z 469.242,A -85,B 0,C 180,E1 -27570.162,E2 -27570.162} C_VEL
LIN {X 0,Y 122.793,Z 471.392,A -85,B 0,C 180,E1 -27572.057,E2 -27572.057} C_VEL
LIN {X 0,Y 121.16,Z 473.426,A -85,B 0,C 180,E1 -27573.419,E2 -27573.419} C_VEL
LIN {X 0,Y 115.922,Z 478.578,A -85,B 0,C 180,E1 -27576.454,E2 -27576.454} C_VEL
LIN {X 0,Y 110.19,Z 483.438,A -85,B 0,C 180,E1 -27579.541,E2 -27579.541} C_VEL
LIN {X 0,Y 102.987,Z 489.092,A -85,B 0,C 180,E1 -27584.23,E2 -27584.23} C_VEL
LIN {X 0,Y 94.814,Z 494.836,A -85,B 0,C 180,E1 -27590.945,E2 -27590.945} C_VEL
LIN {X 0,Y 89.618,Z 498.211,A -85,B 0,C 180,E1 -27596.704,E2 -27596.704} C_VEL
LIN {X 0,Y 84.068,Z 501.635,A -85,B 0,C 180,E1 -27605.291,E2 -27605.291} C_VEL
LIN {X 0,Y 80.38,Z 503.871,A -85,B 0,C 180,E1 -27614.792,E2 -27614.792} C_VEL
LIN {X 0,Y 78.519,Z 504.999,A -85,B 0,C 180,E1 -27624.864,E2 -27624.864} C_VEL
LIN {X 0,Y 78.508,Z 505.007,A -85,B 0,C 180,E1 -27635.135,E2 -27635.135} C_VEL
LIN {X 0,Y 80.38,Z 503.909,A -85,B 0,C 180,E1 -27645.206,E2 -27645.206} C_VEL
LIN {X 0,Y 84.063,Z 501.708,A -85,B 0,C 180,E1 -27654.708,E2 -27654.708} C_VEL
LIN {X 0,Y 89.579,Z 498.33,A -85,B 0,C 180,E1 -27663.311,E2 -27663.311} C_VEL
LIN {X 0,Y 96.635,Z 493.684,A -85,B 0,C 180,E1 -27670.884,E2 -27670.884} C_VEL
LIN {X 0,Y 105.13,Z 487.613,A -85,B 0,C 180,E1 -27677.336,E2 -27677.336} C_VEL
LIN {X 0,Y 113.355,Z 481.05,A -85,B 0,C 180,E1 -27682.231,E2 -27682.231} C_VEL
LIN {X 0,Y 122.278,Z 473.07,A -85,B 0,C 180,E1 -27686.448,E2 -27686.448} C_VEL
LIN {X 0,Y 131.719,Z 463.446,A -85,B 0,C 180,E1 -27690.114,E2 -27690.114} C_VEL
LIN {X 0,Y 140.02,Z 453.595,A -85,B 0,C 180,E1 -27692.968,E2 -27692.968} C_VEL
LIN {X 0,Y 142.491,Z 450.404,A -85,B 0,C 180,E1 -27693.713,E2 -27693.713} C_VEL
LIN {X 0,Y 143.569,Z 448.779,A -85,B 0,C 180,E1 -27694.227,E2 -27694.227} C_VEL
LIN {X 0,Y 144.347,Z 444.491,A -85,B 0,C 180,E1 -27697.679,E2 -27697.679} C_VEL
LIN {X 0,Y 144.732,Z 440.524,A -85,B 0,C 180,E1 -27701.601,E2 -27701.601} C_VEL
LIN {X 0,Y 144.932,Z 437.077,A -85,B 0,C 180,E1 -27705.968,E2 -27705.968} C_VEL
LIN {X 0,Y 144.9,Z 435.445,A -85,B 0,C 180,E1 -27708.813,E2 -27708.813} C_VEL
LIN {X 0,Y 144.981,Z 434.153,A -85,B 0,C 180,E1 -27711.638,E2 -27711.638} C_VEL
LIN {X 0,Y 145.25,Z 432.929,A -85,B 0,C 180,E1 -27717.226,E2 -27717.226} C_VEL
LIN {X 0,Y 145.561,Z 432.751,A -85,B 0,C 180,E1 -27720,E2 -27720} C_VEL
LIN {X 0,Y 145.443,Z 435.167,A -85,B 0,C 180,E1 -27725.546,E2 -27725.546} C_VEL
LIN {X 0,Y 145.59,Z 436.783,A -85,B 0,C 180,E1 -27728.326,E2 -27728.326} C_VEL
LIN {X 0,Y 145.958,Z 439.942,A -85,B 0,C 180,E1 -27732.514,E2 -27732.514} C_VEL
LIN {X 0,Y 146.153,Z 442.149,A -85,B 0,C 180,E1 -27734.803,E2 -27734.803} C_VEL
LIN {X 0,Y 145.139,Z 448.564,A -85,B 0,C 180,E1 -27739.078,E2 -27739.078} C_VEL
LIN {X 0,Y 144.59,Z 451.511,A -85,B 0,C 180,E1 -27740.839,E2 -27740.839} C_VEL
LIN {X 0,Y 138.861,Z 460.817,A -85,B 0,C 180,E1 -27743.462,E2 -27743.462} C_VEL
LIN {X 0,Y 136.425,Z 464.427,A -85,B 0,C 180,E1 -27744.561,E2 -27744.561} C_VEL
LIN {X 0,Y 126.775,Z 475.474,A -85,B 0,C 180,E1 -27747.504,E2 -27747.504} C_VEL
LIN {X 0,Y 118.323,Z 483.955,A -85,B 0,C 180,E1 -27750.543,E2 -27750.543} C_VEL
LIN {X 0,Y 109.118,Z 492.297,A -85,B 0,C 180,E1 -27754.797,E2 -27754.797} C_VEL
LIN {X 0,Y 100.653,Z 499.225,A -85,B 0,C 180,E1 -27759.821,E2 -27759.821} C_VEL
LIN {X 0,Y 92.21,Z 505.696,A -85,B 0,C 180,E1 -27766.691,E2 -27766.691} C_VEL
LIN {X 0,Y 85.339,Z 510.738,A -85,B 0,C 180,E1 -27774.798,E2 -27774.798} C_VEL
LIN {X 0,Y 80.457,Z 514.484,A -85,B 0,C 180,E1 -27784.104,E2 -27784.104} C_VEL
LIN {X 0,Y 77.85,Z 517.018,A -85,B 0,C 180,E1 -27794.288,E2 -27794.288} C_VEL
LIN {X 0,Y 77.666,Z 518.384,A -85,B 0,C 180,E1 -27804.809,E2 -27804.809} C_VEL
LIN {X 0,Y 78.033,Z 518.593,A -85,B 0,C 180,E1 -27810.001,E2 -27810.001} C_VEL
LIN {X 0,Y 77.641,Z 518.372,A -85,B 0,C 180,E1 -27815.313,E2 -27815.313} C_VEL
LIN {X 0,Y 77.857,Z 516.993,A -85,B 0,C 180,E1 -27825.713,E2 -27825.713} C_VEL
LIN {X 0,Y 80.474,Z 514.436,A -85,B 0,C 180,E1 -27835.892,E2 -27835.892} C_VEL
LIN {X 0,Y 85.34,Z 510.657,A -85,B 0,C 180,E1 -27845.204,E2 -27845.204} C_VEL
LIN {X 0,Y 92.227,Z 505.586,A -85,B 0,C 180,E1 -27853.302,E2 -27853.302} C_VEL
LIN {X 0,Y 100.709,Z 499.098,A -85,B 0,C 180,E1 -27860.143,E2 -27860.143} C_VEL
LIN {X 0,Y 106.714,Z 494.246,A -85,B 0,C 180,E1 -27863.78,E2 -27863.78} C_VEL
LIN {X 0,Y 107.326,Z 492.999,A -85,B 0,C 180,E1 -27865.106,E2 -27865.106} C_VEL
LIN {X 0,Y 98.322,Z 490.892,A -85,B 0,C 180,E1 -27874.604,E2 -27874.604} C_VEL
LIN {X 0,Y 92.441,Z 486.881,A -85,B 0,C 180,E1 -27891.254,E2 -27891.254} C_VEL
LIN {X 0,Y 95.973,Z 482.214,A -85,B 0,C 180,E1 -27908.422,E2 -27908.422} C_VEL
LIN {X 0,Y 104.604,Z 477.981,A -85,B 0,C 180,E1 -27919.751,E2 -27919.751} C_VEL
LIN {X 0,Y 119.193,Z 472.355,A -85,B 0,C 180,E1 -27929.785,E2 -27929.785} C_VEL
LIN {X 0,Y 124.453,Z 470.389,A -85,B 0,C 180,E1 -27932.294,E2 -27932.294} C_VEL
LIN {X 0,Y 123.411,Z 471.748,A -85,B 0,C 180,E1 -27933.162,E2 -27933.162} C_VEL
LIN {X 0,Y 113.426,Z 480.811,A -85,B 0,C 180,E1 -27937.813,E2 -27937.813} C_VEL
LIN {X 0,Y 110.19,Z 483.438,A -85,B 0,C 180,E1 -27939.541,E2 -27939.541} C_VEL
LIN {X 0,Y 106.267,Z 486.273,A -85,B 0,C 180,E1 -27941.345,E2 -27941.345} C_VEL
LIN {X 0,Y 98.712,Z 490.636,A -85,B 0,C 180,E1 -27943.983,E2 -27943.983} C_VEL
LIN {X 0,Y 91.243,Z 494.542,A -85,B 0,C 180,E1 -27947.15,E2 -27947.15} C_VEL
LIN {X 0,Y 87.594,Z 496.547,A -85,B 0,C 180,E1 -27949.828,E2 -27949.828} C_VEL
LIN {X 0,Y 80.501,Z 500.687,A -85,B 0,C 180,E1 -27958.41,E2 -27958.41} C_VEL
LIN {X 0,Y 75.348,Z 503.508,A -85,B 0,C 180,E1 -27968.092,E2 -27968.092} C_VEL
LIN {X 0,Y 72.251,Z 505.18,A -85,B 0,C 180,E1 -27978.781,E2 -27978.781} C_VEL
LIN {X 0,Y 71.229,Z 505.754,A -85,B 0,C 180,E1 -27989.999,E2 -27989.999} C_VEL
LIN {X 0,Y 72.239,Z 505.204,A -85,B 0,C 180,E1 -28001.219,E2 -28001.219} C_VEL
LIN {X 0,Y 75.347,Z 503.562,A -85,B 0,C 180,E1 -28011.906,E2 -28011.906} C_VEL
LIN {X 0,Y 80.485,Z 500.781,A -85,B 0,C 180,E1 -28021.595,E2 -28021.595} C_VEL
LIN {X 0,Y 87.398,Z 496.78,A -85,B 0,C 180,E1 -28030.038,E2 -28030.038} C_VEL
LIN {X 0,Y 95.812,Z 491.438,A -85,B 0,C 180,E1 -28037.181,E2 -28037.181} C_VEL
LIN {X 0,Y 105.309,Z 484.613,A -85,B 0,C 180,E1 -28043.21,E2 -28043.21} C_VEL
LIN {X 0,Y 114.462,Z 477.263,A -85,B 0,C 180,E1 -28047.591,E2 -28047.591} C_VEL
LIN {X 0,Y 124.117,Z 468.386,A -85,B 0,C 180,E1 -28051.362,E2 -28051.362} C_VEL
LIN {X 0,Y 133.687,Z 458.085,A -85,B 0,C 180,E1 -28054.622,E2 -28054.622} C_VEL
LIN {X 0,Y 138.435,Z 452.362,A -85,B 0,C 180,E1 -28056.037,E2 -28056.037} C_VEL
LIN {X 0,Y 138.968,Z 451.168,A -85,B 0,C 180,E1 -28056.765,E2 -28056.765} C_VEL
LIN {X 0,Y 139.936,Z 446.779,A -85,B 0,C 180,E1 -28060.948,E2 -28060.948} C_VEL
LIN {X 0,Y 140.474,Z 443.152,A -85,B 0,C 180,E1 -28065.513,E2 -28065.513} C_VEL
LIN {X 0,Y 140.6,Z 441.435,A -85,B 0,C 180,E1 -28068.466,E2 -28068.466} C_VEL
LIN {X 0,Y 140.79,Z 440.121,A -85,B 0,C 180,E1 -28071.387,E2 -28071.387} C_VEL
LIN {X 0,Y 141.045,Z 439.108,A -85,B 0,C 180,E1 -28075.241,E2 -28075.241} C_VEL
LIN {X 0,Y 141.544,Z 438.671,A -85,B 0,C 180,E1 -28080,E2 -28080} C_VEL
LIN {X 0,Y 141.322,Z 441.319,A -85,B 0,C 180,E1 -28085.957,E2 -28085.957} C_VEL
LIN {X 0,Y 141.457,Z 443.823,A -85,B 0,C 180,E1 -28090.014,E2 -28090.014} C_VEL
LIN {X 0,Y 141.604,Z 446.099,A -85,B 0,C 180,E1 -28092.905,E2 -28092.905} C_VEL
LIN {X 0,Y 141.445,Z 447.739,A -85,B 0,C 180,E1 -28094.385,E2 -28094.385} C_VEL
LIN {X 0,Y 139.862,Z 454.434,A -85,B 0,C 180,E1 -28098.945,E2 -28098.945} C_VEL
LIN {X 0,Y 132.676,Z 464.884,A -85,B 0,C 180,E1 -28101.979,E2 -28101.979} C_VEL
LIN {X 0,Y 123.637,Z 474.866,A -85,B 0,C 180,E1 -28104.565,E2 -28104.565} C_VEL
LIN {X 0,Y 113.422,Z 484.592,A -85,B 0,C 180,E1 -28107.998,E2 -28107.998} C_VEL
LIN {X 0,Y 103.846,Z 492.735,A -85,B 0,C 180,E1 -28112.226,E2 -28112.226} C_VEL
LIN {X 0,Y 93.797,Z 500.369,A -85,B 0,C 180,E1 -28118.119,E2 -28118.119} C_VEL
LIN {X 0,Y 85.064,Z 506.478,A -85,B 0,C 180,E1 -28125.392,E2 -28125.392} C_VEL
LIN {X 0,Y 77.731,Z 511.334,A -85,B 0,C 180,E1 -28134.46,E2 -28134.46} C_VEL
LIN {X 0,Y 74.041,Z 513.866,A -85,B 0,C 180,E1 -28141.668,E2 -28141.668} C_VEL
LIN {X 0,Y 70.964,Z 516.401,A -85,B 0,C 180,E1 -28152.717,E2 -28152.717} C_VEL
LIN {X 0,Y 70.566,Z 517.791,A -85,B 0,C 180,E1 -28164.835,E2 -28164.835} C_VEL
LIN {X 0,Y 70.943,Z 517.983,A -85,B 0,C 180,E1 -28170.001,E2 -28170.001} C_VEL
LIN {X 0,Y 70.517,Z 517.761,A -85,B 0,C 180,E1 -28175.721,E2 -28175.721} C_VEL
LIN {X 0,Y 70.971,Z 516.375,A -85,B 0,C 180,E1 -28187.284,E2 -28187.284} C_VEL
LIN {X 0,Y 74.058,Z 513.816,A -85,B 0,C 180,E1 -28198.328,E2 -28198.328} C_VEL
LIN {X 0,Y 79.56,Z 510.036,A -85,B 0,C 180,E1 -28208.198,E2 -28208.198} C_VEL
LIN {X 0,Y 87.123,Z 504.966,A -85,B 0,C 180,E1 -28216.554,E2 -28216.554} C_VEL
LIN {X 0,Y 96.256,Z 498.479,A -85,B 0,C 180,E1 -28223.434,E2 -28223.434} C_VEL
LIN {X 0,Y 99.47,Z 495.949,A -85,B 0,C 180,E1 -28225.582,E2 -28225.582} C_VEL
LIN {X 0,Y 90.304,Z 493.504,A -85,B 0,C 180,E1 -28237.1,E2 -28237.1} C_VEL
LIN {X 0,Y 86.24,Z 489.512,A -85,B 0,C 180,E1 -28255.326,E2 -28255.326} C_VEL
LIN {X 0,Y 92.341,Z 484.788,A -85,B 0,C 180,E1 -28273.199,E2 -28273.199} C_VEL
LIN {X 0,Y 102.698,Z 480.619,A -85,B 0,C 180,E1 -28284.243,E2 -28284.243} C_VEL
LIN {X 0,Y 114.838,Z 476.391,A -85,B 0,C 180,E1 -28291.763,E2 -28291.763} C_VEL
LIN {X 0,Y 113.172,Z 478.162,A -85,B 0,C 180,E1 -28293.032,E2 -28293.032} C_VEL
LIN {X 0,Y 103.433,Z 485.898,A -85,B 0,C 180,E1 -28297.923,E2 -28297.923} C_VEL
LIN {X 0,Y 93.619,Z 492.755,A -85,B 0,C 180,E1 -28304.505,E2 -28304.505} C_VEL
LIN {X 0,Y 87.594,Z 496.547,A -85,B 0,C 180,E1 -28309.828,E2 -28309.828} C_VEL
LIN {X 0,Y 84.078,Z 498.406,A -85,B 0,C 180,E1 -28312.748,E2 -28312.748} C_VEL
LIN {X 0,Y 77.19,Z 501.151,A -85,B 0,C 180,E1 -28317.435,E2 -28317.435} C_VEL
LIN {X 0,Y 71.917,Z 502.991,A -85,B 0,C 180,E1 -28321.8,E2 -28321.8} C_VEL
LIN {X 0,Y 68.918,Z 504.108,A -85,B 0,C 180,E1 -28325.858,E2 -28325.858} C_VEL
LIN {X 0,Y 68.236,Z 504.4,A -85,B 0,C 180,E1 -28327.384,E2 -28327.384} C_VEL
LIN {X 0,Y 65.339,Z 505.788,A -85,B 0,C 180,E1 -28337.576,E2 -28337.576} C_VEL
LIN {X 0,Y 64.163,Z 506.362,A -85,B 0,C 180,E1 -28349.999,E2 -28349.999} C_VEL
LIN {X 0,Y 65.328,Z 505.811,A -85,B 0,C 180,E1 -28362.424,E2 -28362.424} C_VEL
LIN {X 0,Y 68.818,Z 504.171,A -85,B 0,C 180,E1 -28374.109,E2 -28374.109} C_VEL
LIN {X 0,Y 74.541,Z 501.389,A -85,B 0,C 180,E1 -28384.45,E2 -28384.45} C_VEL
LIN {X 0,Y 82.104,Z 497.387,A -85,B 0,C 180,E1 -28393.217,E2 -28393.217} C_VEL
LIN {X 0,Y 91.152,Z 492.044,A -85,B 0,C 180,E1 -28400.444,E2 -28400.444} C_VEL
LIN {X 0,Y 101.222,Z 485.219,A -85,B 0,C 180,E1 -28406.425,E2 -28406.425} C_VEL
LIN {X 0,Y 110.824,Z 477.868,A -85,B 0,C 180,E1 -28410.687,E2 -28410.687} C_VEL
LIN {X 0,Y 120.887,Z 468.988,A -85,B 0,C 180,E1 -28414.305,E2 -28414.305} C_VEL
LIN {X 0,Y 130.757,Z 458.748,A -85,B 0,C 180,E1 -28417.409,E2 -28417.409} C_VEL
LIN {X 0,Y 134.122,Z 454.767,A -85,B 0,C 180,E1 -28418.481,E2 -28418.481} C_VEL
LIN {X 0,Y 135.254,Z 450.84,A -85,B 0,C 180,E1 -28422.669,E2 -28422.669} C_VEL
LIN {X 0,Y 135.668,Z 449.144,A -85,B 0,C 180,E1 -28424.988,E2 -28424.988} C_VEL
LIN {X 0,Y 136.106,Z 446.89,A -85,B 0,C 180,E1 -28428.837,E2 -28428.837} C_VEL
LIN {X 0,Y 136.655,Z 445.024,A -85,B 0,C 180,E1 -28434.096,E2 -28434.096} C_VEL
LIN {X 0,Y 136.954,Z 444.509,A -85,B 0,C 180,E1 -28437.058,E2 -28437.058} C_VEL
LIN {X 0,Y 137.279,Z 444.432,A -85,B 0,C 180,E1 -28440,E2 -28440} C_VEL
LIN {X 0,Y 136.941,Z 447.015,A -85,B 0,C 180,E1 -28445.891,E2 -28445.891} C_VEL
LIN {X 0,Y 136.922,Z 449.778,A -85,B 0,C 180,E1 -28450.349,E2 -28450.349} C_VEL
LIN {X 0,Y 136.83,Z 451.625,A -85,B 0,C 180,E1 -28452.607,E2 -28452.607} C_VEL
LIN {X 0,Y 136.043,Z 454.604,A -85,B 0,C 180,E1 -28454.969,E2 -28454.969} C_VEL
LIN {X 0,Y 135.495,Z 456.374,A -85,B 0,C 180,E1 -28456.246,E2 -28456.246} C_VEL
LIN {X 0,Y 134.918,Z 457.696,A -85,B 0,C 180,E1 -28457.025,E2 -28457.025} C_VEL
LIN {X 0,Y 128.116,Z 466.677,A -85,B 0,C 180,E1 -28459.604,E2 -28459.604} C_VEL
LIN {X 0,Y 117.767,Z 477.25,A -85,B 0,C 180,E1 -28462.334,E2 -28462.334} C_VEL
LIN {X 0,Y 107.307,Z 486.474,A -85,B 0,C 180,E1 -28465.771,E2 -28465.771} C_VEL
LIN {X 0,Y 97.451,Z 494.178,A -85,B 0,C 180,E1 -28470.071,E2 -28470.071} C_VEL
LIN {X 0,Y 87.056,Z 501.415,A -85,B 0,C 180,E1 -28476.169,E2 -28476.169} C_VEL
LIN {X 0,Y 77.958,Z 507.15,A -85,B 0,C 180,E1 -28483.848,E2 -28483.848} C_VEL
LIN {X 0,Y 70.591,Z 511.527,A -85,B 0,C 180,E1 -28493.321,E2 -28493.321} C_VEL
LIN {X 0,Y 65.561,Z 514.658,A -85,B 0,C 180,E1 -28504.611,E2 -28504.611} C_VEL
LIN {X 0,Y 63.384,Z 516.61,A -85,B 0,C 180,E1 -28517.189,E2 -28517.189} C_VEL
LIN {X 0,Y 63.495,Z 517.205,A -85,B 0,C 180,E1 -28524.978,E2 -28524.978} C_VEL
LIN {X 0,Y 63.851,Z 517.373,A -85,B 0,C 180,E1 -28530.001,E2 -28530.001} C_VEL
LIN {X 0,Y 63.385,Z 517.144,A -85,B 0,C 180,E1 -28536.367,E2 -28536.367} C_VEL
LIN {X 0,Y 64.121,Z 515.755,A -85,B 0,C 180,E1 -28549.199,E2 -28549.199} C_VEL
LIN {X 0,Y 67.79,Z 513.195,A -85,B 0,C 180,E1 -28561.224,E2 -28561.224} C_VEL
LIN {X 0,Y 74.039,Z 509.417,A -85,B 0,C 180,E1 -28571.643,E2 -28571.643} C_VEL
LIN {X 0,Y 82.331,Z 504.346,A -85,B 0,C 180,E1 -28580.2,E2 -28580.2} C_VEL
LIN {X 0,Y 89.117,Z 499.935,A -85,B 0,C 180,E1 -28585.176,E2 -28585.176} C_VEL
LIN {X 0,Y 90.56,Z 498.432,A -85,B 0,C 180,E1 -28587.096,E2 -28587.096} C_VEL
LIN {X 0,Y 84.495,Z 496.81,A -85,B 0,C 180,E1 -28595.426,E2 -28595.426} C_VEL
LIN {X 0,Y 79.949,Z 492.963,A -85,B 0,C 180,E1 -28614.957,E2 -28614.957} C_VEL
LIN {X 0,Y 86.233,Z 488.428,A -85,B 0,C 180,E1 -28634.153,E2 -28634.153} C_VEL
LIN {X 0,Y 97.036,Z 484.465,A -85,B 0,C 180,E1 -28645.758,E2 -28645.758} C_VEL
LIN {X 0,Y 105.011,Z 481.91,A -85,B 0,C 180,E1 -28651.057,E2 -28651.057} C_VEL
LIN {X 0,Y 103.293,Z 483.537,A -85,B 0,C 180,E1 -28652.639,E2 -28652.639} C_VEL
LIN {X 0,Y 93.655,Z 490.31,A -85,B 0,C 180,E1 -28658.005,E2 -28658.005} C_VEL
LIN {X 0,Y 84.281,Z 496.055,A -85,B 0,C 180,E1 -28664.862,E2 -28664.862} C_VEL
LIN {X 0,Y 78.159,Z 499.431,A -85,B 0,C 180,E1 -28670.99,E2 -28670.99} C_VEL
LIN {X 0,Y 71.459,Z 502.853,A -85,B 0,C 180,E1 -28680.543,E2 -28680.543} C_VEL
LIN {X 0,Y 68.236,Z 504.4,A -85,B 0,C 180,E1 -28687.384,E2 -28687.384} C_VEL
LIN {X 0,Y 66.024,Z 505.237,A -85,B 0,C 180,E1 -28692.001,E2 -28692.001} C_VEL
LIN {X 0,Y 61.389,Z 506.301,A -85,B 0,C 180,E1 -28699.837,E2 -28699.837} C_VEL
LIN {X 0,Y 58.255,Z 506.809,A -85,B 0,C 180,E1 -28706.885,E2 -28706.885} C_VEL
LIN {X 0,Y 57.197,Z 506.922,A -85,B 0,C 180,E1 -28712.714,E2 -28712.714} C_VEL
LIN {X 0,Y 57.221,Z 506.877,A -85,B 0,C 180,E1 -28714.705,E2 -28714.705} C_VEL
LIN {X 0,Y 58.453,Z 506.418,A -85,B 0,C 180,E1 -28723.913,E2 -28723.913} C_VEL
LIN {X 0,Y 62.435,Z 504.778,A -85,B 0,C 180,E1 -28736.759,E2 -28736.759} C_VEL
LIN {X 0,Y 68.819,Z 501.997,A -85,B 0,C 180,E1 -28747.786,E2 -28747.786} C_VEL
LIN {X 0,Y 77.095,Z 497.995,A -85,B 0,C 180,E1 -28756.825,E2 -28756.825} C_VEL
LIN {X 0,Y 86.819,Z 492.649,A -85,B 0,C 180,E1 -28764.045,E2 -28764.045} C_VEL
LIN {X 0,Y 97.48,Z 485.825,A -85,B 0,C 180,E1 -28769.9,E2 -28769.9} C_VEL
